KUKA KRL program: MyProgram_145().src

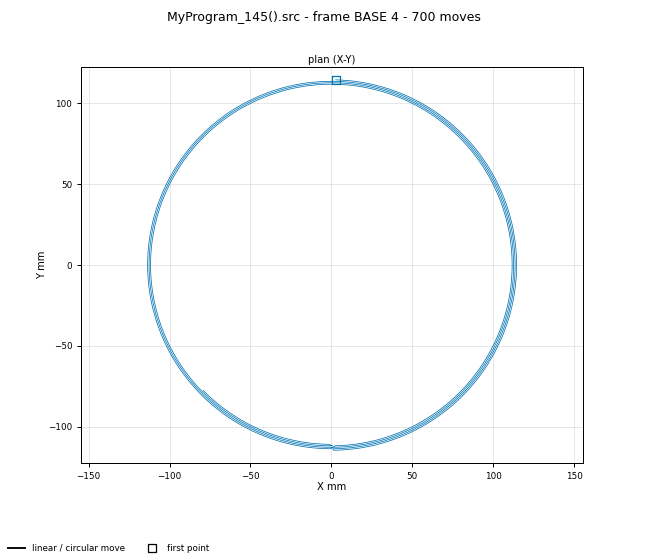
[picture p0: tool path of MyProgram_145().src in frame BASE 4, 700 of 700 moves have a stored position in this frame; points joined in program order, loops and branches not executed]
&ACCESS RVP
&REL 1
&PARAM TEMPLATE = C:\KRC\Roboter\Template\vorgabe
&PARAM EDITMASK = *
DEF MyProgram_145()
; ---- Setting reference (Base) ----
$BASE = BASE_DATA[4]

; --------------------------
; ---- Setting tool (TCP) ----
$TOOL = TOOL_DATA[3]
; --------------------------

$VEL.CP = VEL_APROX_PRINT
Startdeposition()
$VEL.CP = VEL_PRINT
LIN {X 2.5968,Y 114.457,Z 115,A 83.9175,B 24.9348,C -1.8654,E1 25.0049,E2 361.9885} C_DIS
LIN {X 5.4049,Y 114.3588,Z 115,A 82.5188,B 24.9348,C -1.8658,E1 25.0088,E2 363.3858} C_DIS
LIN {X 8.2098,Y 114.1917,Z 115,A 81.1109,B 24.9348,C -1.8657,E1 25.0127,E2 364.7933} C_DIS
LIN {X 10.8808,Y 113.9678,Z 115,A 79.7631,B 24.9348,C -1.8653,E1 25.0164,E2 366.1413} C_DIS
LIN {X 13.803,Y 113.6514,Z 115,A 78.3057,B 24.9348,C -1.8656,E1 25.0205,E2 367.5968} C_DIS
LIN {X 16.588,Y 113.2784,Z 115,A 76.9003,B 24.9348,C -1.8653,E1 25.0244,E2 369.0018} C_DIS
LIN {X 19.573,Y 112.8021,Z 115,A 75.3885,B 24.9348,C -1.8648,E1 25.0285,E2 370.5133} C_DIS
LIN {X 22.3354,Y 112.2877,Z 115,A 73.9836,B 24.9348,C -1.8643,E1 25.0324,E2 371.9177} C_DIS
LIN {X 25.0844,Y 111.7058,Z 115,A 72.5789,B 24.9348,C -1.8636,E1 25.0362,E2 373.3222} C_DIS
LIN {X 27.4876,Y 111.1372,Z 115,A 71.3329,B 24.935,C -1.8625,E1 25.0396,E2 374.569} C_DIS
LIN {X 30.3297,Y 110.3959,Z 115,A 69.8972,B 24.935,C -1.863,E1 25.0434,E2 376.0011} C_DIS
LIN {X 33.234,Y 109.5578,Z 115,A 68.3663,B 24.935,C -1.8611,E1 25.0476,E2 377.534} C_DIS
LIN {X 35.7101,Y 108.7747,Z 115,A 67.0558,B 24.9352,C -1.8596,E1 25.051,E2 378.8456} C_DIS
LIN {X 38.5697,Y 107.7951,Z 115,A 65.5589,B 24.9352,C -1.8589,E1 25.055,E2 380.3411} C_DIS
LIN {X 41.0044,Y 106.8915,Z 115,A 64.249,B 24.9353,C -1.8573,E1 25.0584,E2 381.6521} C_DIS
LIN {X 43.8125,Y 105.7727,Z 115,A 62.7522,B 24.9354,C -1.8564,E1 25.0623,E2 383.1476} C_DIS
LIN {X 46.3951,Y 104.6657,Z 115,A 61.3494,B 24.9355,C -1.855,E1 25.0659,E2 384.5503} C_DIS
LIN {X 48.9498,Y 103.4955,Z 115,A 59.9466,B 24.9356,C -1.8534,E1 25.0694,E2 385.9532} C_DIS
LIN {X 51.4749,Y 102.2631,Z 115,A 58.5442,B 24.9357,C -1.8518,E1 25.0729,E2 387.3557} C_DIS
LIN {X 53.9691,Y 100.969,Z 115,A 57.142,B 24.9358,C -1.8501,E1 25.0764,E2 388.7579} C_DIS
LIN {X 56.2448,Y 99.718,Z 115,A 55.8337,B 24.936,C -1.8479,E1 25.0796,E2 390.0676} C_DIS
LIN {X 58.8584,Y 98.1993,Z 115,A 54.3385,B 24.936,C -1.8464,E1 25.0832,E2 391.5617} C_DIS
LIN {X 60.7218,Y 97.0556,Z 115,A 53.1864,B 24.9364,C -1.8422,E1 25.0859,E2 392.7202} C_DIS
LIN {X 63.1456,Y 95.4964,Z 115,A 51.74,B 24.9366,C -1.8397,E1 25.0893,E2 394.1677} C_DIS
LIN {X 65.9229,Y 93.6033,Z 115,A 50.1344,B 24.9366,C -1.8403,E1 25.093,E2 395.7666} C_DIS
LIN {X 67.7672,Y 92.2743,Z 115,A 48.9337,B 24.9369,C -1.8355,E1 25.0957,E2 396.9743} C_DIS
LIN {X 70.2677,Y 90.3858,Z 115,A 47.4387,B 24.9369,C -1.8359,E1 25.099,E2 398.4629} C_DIS
LIN {X 72.3157,Y 88.7549,Z 115,A 46.1117,B 24.937,C -1.8327,E1 25.1019,E2 399.7924} C_DIS
LIN {X 74.3549,Y 87.0533,Z 115,A 44.7383,B 24.9374,C -1.8281,E1 25.1048,E2 401.1713} C_DIS
LIN {X 76.7265,Y 84.9717,Z 115,A 43.2249,B 24.9374,C -1.8279,E1 25.108,E2 402.6792} C_DIS
LIN {X 78.9438,Y 82.9173,Z 115,A 41.7315,B 24.9375,C -1.8256,E1 25.111,E2 404.1719} C_DIS
LIN {X 80.9549,Y 80.9549,Z 115,A 40.332,B 24.9377,C -1.8229,E1 25.1138,E2 405.5719} C_DIS
LIN {X 82.7695,Y 79.0971,Z 115,A 39.038,B 24.9379,C -1.8203,E1 25.1163,E2 406.8664} C_DIS
LIN {X 84.6857,Y 77.0421,Z 115,A 37.6386,B 24.9381,C -1.8174,E1 25.119,E2 408.2664} C_DIS
LIN {X 86.691,Y 74.7802,Z 115,A 36.1336,B 24.9383,C -1.8143,E1 25.1217,E2 409.7721} C_DIS
LIN {X 88.5001,Y 72.6301,Z 115,A 34.7343,B 24.9385,C -1.8113,E1 25.1242,E2 411.1721} C_DIS
LIN {X 90.1238,Y 70.6034,Z 115,A 33.4288,B 24.9387,C -1.8079,E1 25.1265,E2 412.4795} C_DIS
LIN {X 91.9573,Y 68.2002,Z 115,A 31.9366,B 24.9389,C -1.805,E1 25.129,E2 413.9712} C_DIS
LIN {X 93.6033,Y 65.9229,Z 115,A 30.5381,B 24.9391,C -1.8018,E1 25.1313,E2 415.3705} C_DIS
LIN {X 95.1929,Y 63.6059,Z 115,A 29.1395,B 24.9394,C -1.7986,E1 25.1335,E2 416.7699} C_DIS
LIN {X 96.3998,Y 61.7576,Z 115,A 27.9818,B 24.9397,C -1.7933,E1 25.1352,E2 417.9342} C_DIS
LIN {X 98.1993,Y 58.8584,Z 115,A 26.3429,B 24.9398,C -1.7918,E1 25.1376,E2 419.5682} C_DIS
LIN {X 99.5594,Y 56.5259,Z 115,A 24.9959,B 24.9401,C -1.7884,E1 25.1395,E2 420.9165} C_DIS
LIN {X 100.7076,Y 54.4511,Z 115,A 23.7501,B 24.9405,C -1.7824,E1 25.1412,E2 422.1698} C_DIS
LIN {X 102.1662,Y 51.6645,Z 115,A 22.2423,B 24.9405,C -1.7811,E1 25.1431,E2 423.6728} C_DIS
LIN {X 103.4955,Y 48.9497,Z 115,A 20.7513,B 24.9408,C -1.7777,E1 25.1449,E2 425.1636} C_DIS
LIN {X 104.5678,Y 46.6123,Z 115,A 19.4703,B 24.941,C -1.7743,E1 25.1464,E2 426.4457} C_DIS
LIN {X 105.7727,Y 43.8125,Z 115,A 17.9564,B 24.9413,C -1.7704,E1 25.148,E2 427.9606} C_DIS
LIN {X 106.8161,Y 41.2035,Z 115,A 16.5591,B 24.9415,C -1.7667,E1 25.1495,E2 429.3589} C_DIS
LIN {X 107.7951,Y 38.5697,Z 115,A 15.1617,B 24.9418,C -1.7629,E1 25.1508,E2 430.7574} C_DIS
LIN {X 108.5808,Y 36.2934,Z 115,A 13.9239,B 24.9421,C -1.7578,E1 25.1519,E2 432.0003} C_DIS
LIN {X 109.4947,Y 33.4374,Z 115,A 12.4606,B 24.9423,C -1.7549,E1 25.1531,E2 433.462} C_DIS
LIN {X 110.3313,Y 30.5674,Z 115,A 10.9865,B 24.9425,C -1.7513,E1 25.1543,E2 434.9361} C_DIS
LIN {X 111.0565,Y 27.8182,Z 115,A 9.5735,B 24.9428,C -1.7474,E1 25.1552,E2 436.3502} C_DIS
LIN {X 111.6579,Y 25.2918,Z 115,A 8.2822,B 24.943,C -1.7437,E1 25.1561,E2 437.6427} C_DIS
LIN {X 112.2877,Y 22.3354,Z 115,A 6.7797,B 24.9433,C -1.7394,E1 25.1569,E2 439.1466} C_DIS
LIN {X 112.8021,Y 19.573,Z 115,A 5.3829,B 24.9436,C -1.7354,E1 25.1576,E2 440.5446} C_DIS
LIN {X 113.2159,Y 17.0092,Z 115,A 4.0794,B 24.9438,C -1.7311,E1 25.1582,E2 441.8506} C_DIS
LIN {X 113.6266,Y 14.0145,Z 115,A 2.5896,B 24.9441,C -1.7273,E1 25.1587,E2 443.3406} C_DIS
LIN {X 113.9363,Y 11.2217,Z 115,A 1.193,B 24.9443,C -1.7233,E1 25.1591,E2 444.7385} C_DIS
LIN {X 114.1348,Y 8.9554,Z 115,A 0.0174,B 24.9447,C -1.7179,E1 25.1594,E2 445.9198} C_DIS
LIN {X 114.3379,Y 5.8302,Z 115,A -1.5068,B 24.9449,C -1.7148,E1 25.1596,E2 447.4422} C_DIS
LIN {X 114.4466,Y 3.0225,Z 115,A -2.9032,B 24.9452,C -1.7107,E1 25.1598,E2 448.8399} C_DIS
LIN {X 114.4869,Y 0,Z 115,A -4.3693,B 24.9453,C -1.708,E1 25.1598,E2 450.3038} C_DIS
LIN {X 114.4625,Y -2.2993,Z 115,A -5.5879,B 24.9458,C -1.7011,E1 25.1598,E2 451.5314} C_DIS
LIN {X 114.3588,Y -5.4049,Z 115,A -7.0927,B 24.9459,C -1.6983,E1 25.1596,E2 453.0337} C_DIS
LIN {X 114.1917,Y -8.2098,Z 115,A -8.4892,B 24.9462,C -1.6942,E1 25.1593,E2 454.4317} C_DIS
LIN {X 113.9363,Y -11.2217,Z 115,A -9.9788,B 24.9465,C -1.6903,E1 25.1589,E2 455.9216} C_DIS
LIN {X 113.6693,Y -13.6499,Z 115,A -11.1698,B 24.9466,C -1.6878,E1 25.1585,E2 457.1114} C_DIS
LIN {X 113.2484,Y -16.7988,Z 115,A -12.772,B 24.947,C -1.6821,E1 25.1579,E2 458.7177} C_DIS
LIN {X 112.8021,Y -19.573,Z 115,A -14.1682,B 24.9472,C -1.678,E1 25.1573,E2 460.1154} C_DIS
LIN {X 112.328,Y -22.1263,Z 115,A -15.4716,B 24.9475,C -1.6736,E1 25.1566,E2 461.4214} C_DIS
LIN {X 111.7058,Y -25.0844,Z 115,A -16.9615,B 24.9478,C -1.6698,E1 25.1557,E2 462.9117} C_DIS
LIN {X 111.0565,Y -27.8182,Z 115,A -18.358,B 24.948,C -1.6657,E1 25.1548,E2 464.3097} C_DIS
LIN {X 110.3959,Y -30.3297,Z 115,A -19.6489,B 24.9482,C -1.662,E1 25.1539,E2 465.6021} C_DIS
LIN {X 109.6183,Y -33.0299,Z 115,A -21.058,B 24.9485,C -1.6574,E1 25.1527,E2 467.014} C_DIS
LIN {X 108.7092,Y -35.9127,Z 115,A -22.5483,B 24.9488,C -1.6536,E1 25.1515,E2 468.5046} C_DIS
LIN {X 107.7951,Y -38.5697,Z 115,A -23.9448,B 24.949,C -1.6496,E1 25.1502,E2 469.9027} C_DIS
LIN {X 106.8915,Y -41.0044,Z 115,A -25.236,B 24.9492,C -1.646,E1 25.1489,E2 471.1953} C_DIS
LIN {X 105.7727,Y -43.8125,Z 115,A -26.7388,B 24.9495,C -1.6417,E1 25.1473,E2 472.6998} C_DIS
LIN {X 104.6657,Y -46.3951,Z 115,A -28.1358,B 24.9497,C -1.6379,E1 25.1458,E2 474.0983} C_DIS
LIN {X 103.4955,Y -48.9497,Z 115,A -29.5329,B 24.95,C -1.634,E1 25.1441,E2 475.497} C_DIS
LIN {X 102.3577,Y -51.2841,Z 115,A -30.8241,B 24.9502,C -1.6305,E1 25.1425,E2 476.7895} C_DIS
LIN {X 101.0683,Y -53.7807,Z 115,A -32.234,B 24.9505,C -1.6261,E1 25.1407,E2 478.2023} C_DIS
LIN {X 99.718,Y -56.2448,Z 115,A -33.6189,B 24.9506,C -1.623,E1 25.1388,E2 479.5875} C_DIS
LIN {X 98.1993,Y -58.8584,Z 115,A -35.1221,B 24.9509,C -1.619,E1 25.1367,E2 481.0923} C_DIS
LIN {X 96.8381,Y -61.07,Z 115,A -36.4264,B 24.9511,C -1.615,E1 25.1347,E2 482.3993} C_DIS
LIN {X 95.3102,Y -63.4281,Z 115,A -37.8117,B 24.9513,C -1.612,E1 25.1326,E2 483.7849} C_DIS
LIN {X 93.6033,Y -65.9229,Z 115,A -39.3154,B 24.9515,C -1.6081,E1 25.1302,E2 485.2903} C_DIS
LIN {X 92.0831,Y -68.0284,Z 115,A -40.6198,B 24.9518,C -1.6044,E1 25.1281,E2 486.5972} C_DIS
LIN {X 90.3858,Y -70.2677,Z 115,A -42.0057,B 24.9519,C -1.6015,E1 25.1257,E2 487.9834} C_DIS
LIN {X 88.6342,Y -72.4647,Z 115,A -43.4037,B 24.9521,C -1.5981,E1 25.1233,E2 489.3829} C_DIS
LIN {X 86.691,Y -74.7802,Z 115,A -44.9079,B 24.9524,C -1.5945,E1 25.1205,E2 490.8887} C_DIS
LIN {X 84.9717,Y -76.7265,Z 115,A -46.2006,B 24.9525,C -1.5915,E1 25.1181,E2 492.1827} C_DIS
LIN {X 82.9173,Y -78.9438,Z 115,A -47.7052,B 24.9527,C -1.588,E1 25.1153,E2 493.689} C_DIS
LIN {X 80.9549,Y -80.9549,Z 115,A -49.104,B 24.9529,C -1.5849,E1 25.1125,E2 495.0892} C_DIS
LIN {X 78.9438,Y -82.9173,Z 115,A -50.503,B 24.9531,C -1.5818,E1 25.1097,E2 496.4897} C_DIS
LIN {X 76.8852,Y -84.8297,Z 115,A -51.9019,B 24.9533,C -1.5788,E1 25.1068,E2 497.8901} C_DIS
LIN {X 74.9406,Y -86.5509,Z 115,A -53.1952,B 24.9535,C -1.5761,E1 25.1041,E2 499.1846} C_DIS
LIN {X 72.6302,Y -88.5001,Z 115,A -54.701,B 24.9536,C -1.573,E1 25.1009,E2 500.6919} C_DIS
LIN {X 70.4364,Y -90.2559,Z 115,A -56.1002,B 24.9538,C -1.5702,E1 25.0978,E2 502.0925} C_DIS
LIN {X 68.3704,Y -91.8294,Z 115,A -57.4068,B 24.954,C -1.5671,E1 25.0949,E2 503.4016} C_DIS
LIN {X 66.0962,Y -93.4796,Z 115,A -58.7941,B 24.9541,C -1.5651,E1 25.0917,E2 504.7889} C_DIS
LIN {X 63.6059,Y -95.1929,Z 115,A -60.3003,B 24.9543,C -1.5623,E1 25.0882,E2 506.2966} C_DIS
LIN {X 61.4298,Y -96.6102,Z 115,A -61.6073,B 24.9544,C -1.5594,E1 25.0852,E2 507.6061} C_DIS
LIN {X 58.8584,Y -98.1993,Z 115,A -63.1013,B 24.9546,C -1.5574,E1 25.0816,E2 509.1002} C_DIS
LIN {X 56.4307,Y -99.6142,Z 115,A -64.5018,B 24.9546,C -1.5551,E1 25.0782,E2 510.5019} C_DIS
LIN {X 52.726,Y -101.6237,Z 115,A -66.6037,B 24.9549,C -1.5518,E1 25.073,E2 512.6057} C_DIS
LIN {X 50.2161,Y -102.8871,Z 115,A -68.0047,B 24.955,C -1.5497,E1 25.0695,E2 514.0079} C_DIS
LIN {X 47.8691,Y -103.9986,Z 115,A -69.3001,B 24.9551,C -1.5478,E1 25.0662,E2 515.3044} C_DIS
LIN {X 45.3024,Y -105.142,Z 115,A -70.7144,B 24.9553,C -1.5453,E1 25.0626,E2 516.7212} C_DIS
LIN {X 42.7084,Y -106.2221,Z 115,A -72.1165,B 24.9553,C -1.5435,E1 25.059,E2 518.1244} C_DIS
LIN {X 39.8896,Y -107.3137,Z 115,A -73.6122,B 24.9554,C -1.5421,E1 25.0551,E2 519.62} C_DIS
LIN {X 37.4449,Y -108.1898,Z 115,A -74.9078,B 24.9555,C -1.5407,E1 25.0517,E2 520.9166} C_DIS
LIN {X 34.7785,Y -109.0762,Z 115,A -76.3108,B 24.9556,C -1.5391,E1 25.0479,E2 522.3206} C_DIS
LIN {X 31.887,Y -109.9574,Z 115,A -77.8197,B 24.9557,C -1.5375,E1 25.0439,E2 523.8307} C_DIS
LIN {X 29.179,Y -110.7068,Z 115,A -79.2228,B 24.9557,C -1.5361,E1 25.0401,E2 525.2348} C_DIS
LIN {X 26.6601,Y -111.3391,Z 115,A -80.5196,B 24.9559,C -1.535,E1 25.0366,E2 526.5324} C_DIS
LIN {X 23.9197,Y -111.9598,Z 115,A -81.923,B 24.9559,C -1.5338,E1 25.0328,E2 527.9368} C_DIS
LIN {X 20.9558,Y -112.5534,Z 115,A -83.4333,B 24.9559,C -1.5326,E1 25.0286,E2 529.4481} C_DIS
LIN {X 18.3973,Y -112.9986,Z 115,A -84.7433,B 24.9561,C -1.5311,E1 25.025,E2 530.7601} C_DIS
LIN {X 15.6186,Y -113.4161,Z 115,A -86.1372,B 24.9561,C -1.5307,E1 25.0212,E2 532.1538} C_DIS
LIN {X 12.6191,Y -113.79,Z 115,A -87.6457,B 24.9561,C -1.53,E1 25.017,E2 533.663} C_DIS
LIN {X 10.0348,Y -114.0459,Z 115,A -88.9441,B 24.9561,C -1.5293,E1 25.0134,E2 534.9621} C_DIS
LIN {X 7.0205,Y -114.2721,Z 115,A -90.4554,B 24.9562,C -1.5287,E1 25.0091,E2 536.4742} C_DIS
LIN {X 4.214,Y -114.41,Z 115,A -91.8604,B 24.9562,C -1.5282,E1 25.0052,E2 537.8799} C_DIS
LIN {X 1.4049,Y -114.479,Z 115,A -93.2656,B 24.9562,C -1.5279,E1 25.0013,E2 539.2858} C_DIS
LIN {X 1.4049,Y -114.479,Z 115,A -93.2656,B 24.9562,C -1.5279,E1 25.0013,E2 539.2858} C_DIS
Enddeposition()
LIN {X 0.793,Y -113.5682,Z 115,A -93.0605,B 24.954,C -1.5662,E1 25.0021,E2 538.9899} C_DIS
Startdeposition()
$VEL.CP = VEL_PRINT
LIN {X 3.5216,Y -113.5178,Z 115,A -91.1293,B 24.9526,C -1.591,E1 25.0077,E2 537.0003} C_DIS
LIN {X 6.9982,Y -113.3576,Z 115,A -89.1991,B 24.9521,C -1.5995,E1 25.0131,E2 535.0508} C_DIS
LIN {X 11.2037,Y -113.0202,Z 115,A -87.4324,B 24.953,C -1.5845,E1 25.0179,E2 533.3206} C_DIS
LIN {X 15.2462,Y -112.546,Z 115,A -84.7536,B 24.9512,C -1.6138,E1 25.0255,E2 530.5747} C_DIS
LIN {X 20.5071,Y -111.7064,Z 115,A -82.954,B 24.9535,C -1.5762,E1 25.0302,E2 528.866} C_DIS
LIN {X 23.3283,Y -111.1518,Z 115,A -81.5254,B 24.9535,C -1.5765,E1 25.0341,E2 527.4385} C_DIS
LIN {X 26.2423,Y -110.5012,Z 115,A -79.8314,B 24.9529,C -1.5863,E1 25.0388,E2 525.7237} C_DIS
LIN {X 30.1207,Y -109.5066,Z 115,A -78.0115,B 24.9533,C -1.5795,E1 25.0437,E2 523.9227} C_DIS
LIN {X 33.4764,Y -108.5267,Z 115,A -76.2704,B 24.9532,C -1.5806,E1 25.0483,E2 522.1821} C_DIS
LIN {X 36.5165,Y -107.5421,Z 115,A -74.492,B 24.9526,C -1.59,E1 25.0531,E2 520.3848} C_DIS
LIN {X 41.5359,Y -105.7046,Z 115,A -71.5463,B 24.9517,C -1.605,E1 25.0608,E2 517.41} C_DIS
LIN {X 44.5412,Y -104.4748,Z 115,A -70.157,B 24.9523,C -1.5961,E1 25.0644,E2 516.045} C_DIS
LIN {X 48.1845,Y -102.8446,Z 115,A -68.3364,B 24.9526,C -1.5905,E1 25.0689,E2 514.2422} C_DIS
LIN {X 51.1511,Y -101.4032,Z 115,A -66.6992,B 24.9526,C -1.592,E1 25.073,E2 512.6057} C_DIS
LIN {X 54.0223,Y -99.9014,Z 115,A -64.9679,B 24.9521,C -1.5993,E1 25.0773,E2 510.8623} C_DIS
LIN {X 56.7874,Y -98.3561,Z 115,A -63.465,B 24.9521,C -1.5978,E1 25.081,E2 509.3673} C_DIS
LIN {X 59.5307,Y -96.7221,Z 115,A -61.5707,B 24.9512,C -1.6138,E1 25.0856,E2 507.4412} C_DIS
LIN {X 63.3856,Y -94.2395,Z 115,A -59.4229,B 24.9514,C -1.6108,E1 25.0905,E2 505.3076} C_DIS
LIN {X 66.4794,Y -92.0846,Z 115,A -57.6419,B 24.9514,C -1.6092,E1 25.0946,E2 503.5366} C_DIS
LIN {X 69.0541,Y -90.1684,Z 115,A -56.0169,B 24.9513,C -1.6129,E1 25.0982,E2 501.9086} C_DIS
LIN {X 71.7186,Y -88.0636,Z 115,A -54.1829,B 24.9507,C -1.6223,E1 25.1022,E2 500.0594} C_DIS
LIN {X 74.7011,Y -85.5478,Z 115,A -52.3131,B 24.9507,C -1.6223,E1 25.1062,E2 498.1969} C_DIS
LIN {X 77.2866,Y -83.2222,Z 115,A -50.4101,B 24.95,C -1.6332,E1 25.1101,E2 496.2757} C_DIS
LIN {X 79.9158,Y -80.698,Z 115,A -48.7126,B 24.9501,C -1.6312,E1 25.1135,E2 494.5901} C_DIS
LIN {X 82.5394,Y -78.0129,Z 115,A -46.8265,B 24.9499,C -1.6356,E1 25.1171,E2 492.7018} C_DIS
LIN {X 84.8762,Y -75.4643,Z 115,A -45.1773,B 24.9499,C -1.6356,E1 25.1202,E2 491.0597} C_DIS
LIN {X 87.1423,Y -72.8355,Z 115,A -43.3428,B 24.9493,C -1.6441,E1 25.1236,E2 489.2136} C_DIS
LIN {X 89.4592,Y -69.972,Z 115,A -41.4045,B 24.9488,C -1.6528,E1 25.1269,E2 487.2639} C_DIS
LIN {X 91.6183,Y -67.1176,Z 115,A -39.7048,B 24.9488,C -1.6529,E1 25.1298,E2 485.5722} C_DIS
LIN {X 93.3527,Y -64.6838,Z 115,A -38.187,B 24.9485,C -1.6576,E1 25.1322,E2 484.0508} C_DIS
LIN {X 95.0825,Y -62.1147,Z 115,A -36.7548,B 24.9486,C -1.6559,E1 25.1344,E2 482.6296} C_DIS
LIN {X 96.7961,Y -59.4091,Z 115,A -34.9771,B 24.9479,C -1.6681,E1 25.137,E2 480.8321} C_DIS
LIN {X 98.7922,Y -56.0286,Z 115,A -32.9319,B 24.9473,C -1.677,E1 25.1399,E2 478.7767} C_DIS
LIN {X 100.7462,Y -52.4329,Z 115,A -31.1232,B 24.9477,C -1.6712,E1 25.1423,E2 476.9912} C_DIS
LIN {X 102.1239,Y -49.6963,Z 115,A -29.3014,B 24.9466,C -1.6887,E1 25.1445,E2 475.1377} C_DIS
LIN {X 104.0236,Y -45.5832,Z 115,A -27.1729,B 24.9466,C -1.6884,E1 25.147,E2 473.0215} C_DIS
LIN {X 105.434,Y -42.2225,Z 115,A -25.4888,B 24.9466,C -1.6868,E1 25.1487,E2 471.3503} C_DIS
LIN {X 106.9636,Y -38.1818,Z 115,A -23.3424,B 24.9463,C -1.6921,E1 25.1508,E2 469.2036} C_DIS
LIN {X 108.0365,Y -35.0258,Z 115,A -21.6182,B 24.9459,C -1.6994,E1 25.1524,E2 467.4719} C_DIS
LIN {X 109.0809,Y -31.6306,Z 115,A -19.8607,B 24.9456,C -1.7035,E1 25.1538,E2 465.7149} C_DIS
LIN {X 110.0465,Y -28.0802,Z 115,A -17.9109,B 24.945,C -1.7138,E1 25.1552,E2 463.7518} C_DIS
LIN {X 110.7958,Y -24.9668,Z 115,A -16.4113,B 24.945,C -1.7136,E1 25.1561,E2 462.2615} C_DIS
LIN {X 111.3099,Y -22.5582,Z 115,A -15.0009,B 24.9442,C -1.7255,E1 25.1569,E2 460.8313} C_DIS
LIN {X 112.007,Y -18.7917,Z 115,A -13.1014,B 24.9439,C -1.7302,E1 25.1578,E2 458.9318} C_DIS
LIN {X 112.5769,Y -15.0105,Z 115,A -11.227,B 24.9437,C -1.7339,E1 25.1586,E2 457.0597} C_DIS
LIN {X 113.2173,Y -8.9741,Z 115,A -8.4018,B 24.9437,C -1.7327,E1 25.1594,E2 454.2539} C_DIS
LIN {X 113.3861,Y -6.5058,Z 115,A -6.9816,B 24.9429,C -1.7448,E1 25.1596,E2 452.8136} C_DIS
LIN {X 113.5363,Y -2.917,Z 115,A -4.3528,B 24.94,C -1.7892,E1 25.1598,E2 450.0958} C_DIS
LIN {X 113.5471,Y 2.4173,Z 115,A -2.7769,B 24.9429,C -1.7455,E1 25.1598,E2 448.6324} C_DIS
LIN {X 113.2765,Y 8.2121,Z 115,A 0.436,B 24.9414,C -1.7683,E1 25.1593,E2 445.3849} C_DIS
LIN {X 112.7669,Y 13.5054,Z 115,A 2.9476,B 24.9414,C -1.7689,E1 25.1586,E2 442.8867} C_DIS
LIN {X 112.3726,Y 16.4724,Z 115,A 4.6823,B 24.9403,C -1.7842,E1 25.1579,E2 441.1262} C_DIS
LIN {X 111.7823,Y 20.0848,Z 115,A 6.415,B 24.9403,C -1.7847,E1 25.157,E2 439.4023} C_DIS
LIN {X 111.1336,Y 23.4171,Z 115,A 8.0257,B 24.9403,C -1.7853,E1 25.1561,E2 437.7996} C_DIS
LIN {X 110.3519,Y 26.8541,Z 115,A 9.8366,B 24.9398,C -1.7924,E1 25.155,E2 435.9825} C_DIS
LIN {X 109.5022,Y 30.1371,Z 115,A 11.4761,B 24.9397,C -1.7944,E1 25.1538,E2 434.3479} C_DIS
LIN {X 108.7794,Y 32.6475,Z 115,A 12.7391,B 24.9396,C -1.7959,E1 25.1528,E2 433.0885} C_DIS
LIN {X 107.8376,Y 35.64,Z 115,A 14.5381,B 24.9385,C -1.8107,E1 25.1513,E2 431.2648} C_DIS
LIN {X 106.4359,Y 39.6278,Z 115,A 17.2456,B 24.9363,C -1.8439,E1 25.1486,E2 428.4941} C_DIS
LIN {X 104.7174,Y 43.9657,Z 115,A 19.028,B 24.9376,C -1.8241,E1 25.1467,E2 426.7682} C_DIS
LIN {X 102.9135,Y 48.0365,Z 115,A 21.1776,B 24.9375,C -1.8261,E1 25.1443,E2 424.6255} C_DIS
LIN {X 101.1901,Y 51.568,Z 115,A 23.0853,B 24.9373,C -1.8282,E1 25.1419,E2 422.7229} C_DIS
LIN {X 99.69,Y 54.4122,Z 115,A 24.8126,B 24.9367,C -1.8376,E1 25.1396,E2 420.9827} C_DIS
LIN {X 97.6246,Y 58.0362,Z 115,A 26.897,B 24.9364,C -1.8423,E1 25.1367,E2 418.8978} C_DIS
LIN {X 95.8022,Y 60.9983,Z 115,A 28.5559,B 24.9364,C -1.8426,E1 25.1342,E2 417.2468} C_DIS
LIN {X 93.9892,Y 63.7552,Z 115,A 30.2244,B 24.936,C -1.8471,E1 25.1316,E2 415.5759} C_DIS
LIN {X 91.8075,Y 66.8592,Z 115,A 32.1034,B 24.9358,C -1.8503,E1 25.1286,E2 413.6984} C_DIS
LIN {X 89.2992,Y 70.1743,Z 115,A 34.2418,B 24.9353,C -1.8573,E1 25.1249,E2 411.5536} C_DIS
LIN {X 86.9459,Y 73.0718,Z 115,A 35.9983,B 24.9354,C -1.856,E1 25.1218,E2 409.8084} C_DIS
LIN {X 85.1265,Y 75.1835,Z 115,A 37.8359,B 24.9338,C -1.8789,E1 25.1183,E2 407.9248} C_DIS
LIN {X 82.9605,Y 77.5651,Z 115,A 38.8497,B 24.9355,C -1.8548,E1 25.1165,E2 406.9725} C_DIS
LIN {X 81.1764,Y 79.4315,Z 115,A 40.4567,B 24.9343,C -1.8714,E1 25.1133,E2 405.333} C_DIS
LIN {X 78.5548,Y 82.0241,Z 115,A 42.3562,B 24.9339,C -1.8772,E1 25.1095,E2 403.4279} C_DIS
LIN {X 76.3037,Y 84.1241,Z 115,A 43.7221,B 24.9343,C -1.8719,E1 25.1068,E2 402.0801} C_DIS
LIN {X 74.383,Y 85.8256,Z 115,A 44.9967,B 24.9342,C -1.8735,E1 25.1041,E2 400.8066} C_DIS
LIN {X 71.7145,Y 88.067,Z 115,A 46.7426,B 24.934,C -1.8764,E1 25.1003,E2 399.0607} C_DIS
LIN {X 69.2353,Y 90.0287,Z 115,A 48.4361,B 24.9335,C -1.8838,E1 25.0966,E2 397.3559} C_DIS
LIN {X 66.661,Y 91.9526,Z 115,A 50.3108,B 24.9325,C -1.898,E1 25.0923,E2 395.4542} C_DIS
LIN {X 61.7781,Y 95.3017,Z 115,A 52.8464,B 24.9336,C -1.8826,E1 25.0865,E2 392.9634} C_DIS
LIN {X 59.1525,Y 96.9521,Z 115,A 54.5541,B 24.9329,C -1.8915,E1 25.0824,E2 391.2403} C_DIS
LIN {X 55.9057,Y 98.8616,Z 115,A 56.5872,B 24.9323,C -1.9001,E1 25.0775,E2 389.1929} C_DIS
LIN {X 52.271,Y 100.8308,Z 115,A 59.5639,B 24.9292,C -1.9428,E1 25.0699,E2 386.1234} C_DIS
LIN {X 46.742,Y 103.5079,Z 115,A 61.52,B 24.9326,C -1.8955,E1 25.0652,E2 384.2843} C_DIS
LIN {X 44.5083,Y 104.4887,Z 115,A 62.9545,B 24.9319,C -1.9058,E1 25.0615,E2 382.8287} C_DIS
LIN {X 41.3685,Y 105.7703,Z 115,A 64.594,B 24.932,C -1.9044,E1 25.0572,E2 381.1963} C_DIS
LIN {X 38.3334,Y 106.9094,Z 115,A 66.2855,B 24.9317,C -1.9084,E1 25.0528,E2 379.4989} C_DIS
LIN {X 35.2317,Y 107.9699,Z 115,A 67.8646,B 24.9319,C -1.9065,E1 25.0486,E2 377.9273} C_DIS
LIN {X 32.0949,Y 108.9433,Z 115,A 69.5697,B 24.9316,C -1.9098,E1 25.044,E2 376.2173} C_DIS
LIN {X 28.9079,Y 109.8337,Z 115,A 71.0773,B 24.932,C -1.9038,E1 25.04,E2 374.7263} C_DIS
LIN {X 26.7238,Y 110.3837,Z 115,A 72.3303,B 24.9316,C -1.9096,E1 25.0366,E2 373.4614} C_DIS
LIN {X 23.5774,Y 111.1,Z 115,A 73.847,B 24.9319,C -1.9056,E1 25.0325,E2 371.9563} C_DIS
LIN {X 19.753,Y 111.842,Z 115,A 75.8698,B 24.9317,C -1.9089,E1 25.0269,E2 369.928} C_DIS
LIN {X 16.0692,Y 112.4299,Z 115,A 78.0906,B 24.9306,C -1.9241,E1 25.0207,E2 367.6731} C_DIS
LIN {X 11.714,Y 112.9667,Z 115,A 80.2368,B 24.9308,C -1.9215,E1 25.0147,E2 365.5345} C_DIS
LIN {X 7.3617,Y 113.3339,Z 115,A 82.1205,B 24.9318,C -1.9079,E1 25.0096,E2 363.6841} C_DIS
LIN {X 1.1044,Y 113.5677,Z 115,A 85.1447,B 24.9322,C -1.9018,E1 25.0012,E2 360.6751} C_DIS
LIN {X -5.6869,Y 113.4314,Z 115,A 88.6544,B 24.932,C -1.9042,E1 24.9914,E2 357.1591} C_DIS
LIN {X -12.5625,Y 112.8773,Z 115,A 92.1705,B 24.932,C -1.9041,E1 24.9816,E2 353.6418} C_DIS
LIN {X -15.4607,Y 112.5163,Z 115,A 93.7976,B 24.9316,C -1.9097,E1 24.977,E2 352.0001} C_DIS
LIN {X -18.9323,Y 111.9835,Z 115,A 95.4868,B 24.932,C -1.9049,E1 24.9724,E2 350.3206} C_DIS
LIN {X -22.6369,Y 111.2938,Z 115,A 97.4268,B 24.932,C -1.905,E1 24.9671,E2 348.3783} C_DIS
LIN {X -26.2566,Y 110.4977,Z 115,A 99.2119,B 24.9323,C -1.8998,E1 24.9623,E2 346.6034} C_DIS
LIN {X -29.7238,Y 109.6138,Z 115,A 101.1437,B 24.9321,C -1.9033,E1 24.957,E2 344.6604} C_DIS
LIN {X -33.7888,Y 108.4298,Z 115,A 103.2853,B 24.9322,C -1.9011,E1 24.9513,E2 342.5204} C_DIS
LIN {X -37.4761,Y 107.2112,Z 115,A 105.2615,B 24.9324,C -1.8994,E1 24.9461,E2 340.5444} C_DIS
LIN {X -41.4151,Y 105.752,Z 115,A 107.3253,B 24.9327,C -1.8943,E1 24.9407,E2 338.4885} C_DIS
LIN {X -45.2042,Y 104.1888,Z 115,A 109.2418,B 24.9334,C -1.885,E1 24.9358,E2 336.5895} C_DIS
LIN {X -47.5976,Y 103.1178,Z 115,A 110.6962,B 24.9331,C -1.8884,E1 24.9321,E2 335.1235} C_DIS
LIN {X -53.0774,Y 100.4067,Z 115,A 113.9148,B 24.9331,C -1.8889,E1 24.9241,E2 331.8953} C_DIS
LIN {X -56.5974,Y 98.4653,Z 115,A 115.8907,B 24.9335,C -1.8832,E1 24.9192,E2 329.9271} C_DIS
LIN {X -60.6035,Y 96.0529,Z 115,A 118.1284,B 24.9342,C -1.8738,E1 24.914,E2 327.7049} C_DIS
LIN {X -63.2127,Y 94.3565,Z 115,A 119.7424,B 24.9342,C -1.8725,E1 24.9102,E2 326.0885} C_DIS
LIN {X -65.9791,Y 92.4416,Z 115,A 121.5286,B 24.9342,C -1.8727,E1 24.9061,E2 324.2957} C_DIS
LIN {X -68.5003,Y 90.5899,Z 115,A 123.0471,B 24.9347,C -1.867,E1 24.9027,E2 322.7855} C_DIS
LIN {X -71.1466,Y 88.5272,Z 115,A 124.6224,B 24.9353,C -1.8585,E1 24.8993,E2 321.2245} C_DIS
LIN {X -72.8647,Y 87.118,Z 115,A 125.8209,B 24.9353,C -1.8592,E1 24.8967,E2 320.0198} C_DIS
LIN {X -74.7298,Y 85.5227,Z 115,A 127.2065,B 24.935,C -1.8623,E1 24.8937,E2 318.6213} C_DIS
LIN {X -77.3644,Y 83.1493,Z 115,A 129.0946,B 24.935,C -1.8621,E1 24.8899,E2 316.726} C_DIS
LIN {X -80.3903,Y 80.2273,Z 115,A 130.9762,B 24.936,C -1.8473,E1 24.8862,E2 314.8718} C_DIS
LIN {X -82.0223,Y 78.5568,Z 115,A 132.1783,B 24.9362,C -1.8454,E1 24.8838,E2 313.6692} C_DIS
LIN {X -83.6587,Y 76.8108,Z 115,A 133.5393,B 24.9359,C -1.8485,E1 24.8812,E2 312.2947} C_DIS
LIN {X -85.8919,Y 74.3071,Z 115,A 135.1233,B 24.9366,C -1.8398,E1 24.8783,E2 310.7243} C_DIS
LIN {X -88.1599,Y 71.5998,Z 115,A 137.0204,B 24.9366,C -1.8398,E1 24.8749,E2 308.8185} C_DIS
LIN {X -89.8764,Y 69.433,Z 115,A 138.4651,B 24.9366,C -1.838,E1 24.8725,E2 307.3712} C_DIS
LIN {X -92.3919,Y 66.0488,Z 115,A 140.5171,B 24.9373,C -1.8292,E1 24.8691,E2 305.3303} C_DIS
LIN {X -94.9972,Y 62.2441,Z 115,A 143.0368,B 24.9373,C -1.8304,E1 24.8651,E2 302.7951} C_DIS
LIN {X -97.6334,Y 58.0213,Z 115,A 145.5732,B 24.9376,C -1.8242,E1 24.8615,E2 300.2606} C_DIS
LIN {X -100.0382,Y 53.7701,Z 115,A 147.7983,B 24.9388,C -1.8074,E1 24.8585,E2 298.0637} C_DIS
LIN {X -101.6163,Y 50.7238,Z 115,A 149.5615,B 24.939,C -1.8035,E1 24.8563,E2 296.3004} C_DIS
LIN {X -103.0763,Y 47.6869,Z 115,A 151.224,B 24.9395,C -1.7969,E1 24.8543,E2 294.6446} C_DIS
LIN {X -104.5463,Y 44.3717,Z 115,A 153.4502,B 24.9388,C -1.8071,E1 24.8518,E2 292.3817} C_DIS
LIN {X -106.3238,Y 39.9255,Z 115,A 155.5265,B 24.9402,C -1.7861,E1 24.8497,E2 290.3439} C_DIS
LIN {X -107.4582,Y 36.7652,Z 115,A 157.8104,B 24.939,C -1.8043,E1 24.8476,E2 288.0036} C_DIS
LIN {X -108.6452,Y 33.0938,Z 115,A 159.1494,B 24.941,C -1.7739,E1 24.8465,E2 286.7293} C_DIS
LIN {X -109.4371,Y 30.3739,Z 115,A 160.9454,B 24.9404,C -1.7839,E1 24.8451,E2 284.899} C_DIS
LIN {X -110.3649,Y 26.8009,Z 115,A 162.5325,B 24.9415,C -1.7671,E1 24.8441,E2 283.3429} C_DIS
LIN {X -111.0575,Y 23.772,Z 115,A 164.0567,B 24.9419,C -1.7603,E1 24.8432,E2 281.8259} C_DIS
LIN {X -111.6428,Y 20.8559,Z 115,A 165.8197,B 24.9416,C -1.7659,E1 24.8422,E2 280.0392} C_DIS
LIN {X -112.1949,Y 17.6376,Z 115,A 167.2848,B 24.9424,C -1.7533,E1 24.8416,E2 278.5952} C_DIS
LIN {X -112.6393,Y 14.5283,Z 115,A 168.9357,B 24.9425,C -1.7508,E1 24.841,E2 276.9404} C_DIS
LIN {X -113.0125,Y 11.2767,Z 115,A 170.6947,B 24.9426,C -1.7497,E1 24.8404,E2 275.1735} C_DIS
LIN {X -113.2977,Y 7.8984,Z 115,A 172.3163,B 24.9432,C -1.7407,E1 24.8401,E2 273.5639} C_DIS
LIN {X -113.4806,Y 4.5744,Z 115,A 174.0587,B 24.9434,C -1.7377,E1 24.8399,E2 271.8181} C_DIS
LIN {X -113.5702,Y 0.7165,Z 115,A 176.0092,B 24.9438,C -1.7315,E1 24.8398,E2 269.8705} C_DIS
LIN {X -113.5239,Y -3.3225,Z 115,A 178.0504,B 24.9442,C -1.725,E1 24.8398,E2 267.8324} C_DIS
LIN {X -113.3332,Y -7.373,Z 115,A -179.933,B 24.9447,C -1.7173,E1 24.8402,E2 265.8222} C_DIS
LIN {X -113.0459,Y -10.9348,Z 115,A -178.1846,B 24.9452,C -1.7093,E1 24.8406,E2 264.0823} C_DIS
LIN {X -112.7864,Y -13.3391,Z 115,A -176.9395,B 24.9454,C -1.7064,E1 24.841,E2 262.8367} C_DIS
LIN {X -112.3452,Y -16.6648,Z 115,A -175.0424,B 24.9453,C -1.7092,E1 24.8418,E2 260.9217} C_DIS
LIN {X -111.8036,Y -19.9665,Z 115,A -173.4065,B 24.9457,C -1.7018,E1 24.8426,E2 259.2937} C_DIS
LIN {X -111.145,Y -23.3614,Z 115,A -171.6451,B 24.946,C -1.6969,E1 24.8435,E2 257.5334} C_DIS
LIN {X -110.3339,Y -26.9281,Z 115,A -169.8542,B 24.9465,C -1.6891,E1 24.8447,E2 255.7508} C_DIS
LIN {X -108.2801,Y -34.2719,Z 115,A -165.3888,B 24.9457,C -1.7021,E1 24.8483,E2 251.2286} C_DIS
LIN {X -106.9164,Y -38.3143,Z 115,A -163.9116,B 24.9478,C -1.6685,E1 24.8496,E2 249.8231} C_DIS
LIN {X -106.0683,Y -40.6001,Z 115,A -162.6951,B 24.9481,C -1.6643,E1 24.8507,E2 248.6097} C_DIS
LIN {X -105.2093,Y -42.7748,Z 115,A -161.472,B 24.9481,C -1.6626,E1 24.852,E2 247.3838} C_DIS
LIN {X -103.9172,Y -45.8273,Z 115,A -159.5857,B 24.948,C -1.6664,E1 24.8541,E2 245.4781} C_DIS
LIN {X -102.1287,Y -49.6863,Z 115,A -157.5633,B 24.9487,C -1.6553,E1 24.8565,E2 243.4711} C_DIS
LIN {X -100.0587,Y -53.7323,Z 115,A -155.2087,B 24.9489,C -1.6514,E1 24.8596,E2 241.1132} C_DIS
LIN {X -98.2969,Y -56.8904,Z 115,A -153.4798,B 24.9494,C -1.6426,E1 24.8619,E2 239.3962} C_DIS
LIN {X -96.9399,Y -59.1725,Z 115,A -152.0842,B 24.9495,C -1.6413,E1 24.864,E2 237.9965} C_DIS
LIN {X -95.405,Y -61.6172,Z 115,A -150.681,B 24.9499,C -1.6354,E1 24.8661,E2 236.6005} C_DIS
LIN {X -93.5701,Y -64.3709,Z 115,A -149.0489,B 24.9502,C -1.6296,E1 24.8686,E2 234.974} C_DIS
LIN {X -91.6717,Y -67.0446,Z 115,A -147.3589,B 24.9504,C -1.6269,E1 24.8714,E2 233.2822} C_DIS
LIN {X -89.4421,Y -69.9935,Z 115,A -145.5182,B 24.9507,C -1.6213,E1 24.8745,E2 231.446} C_DIS
LIN {X -87.9082,Y -71.9104,Z 115,A -144.2034,B 24.9507,C -1.6215,E1 24.8768,E2 230.1247} C_DIS
LIN {X -82.6332,Y -77.9132,Z 115,A -140.0978,B 24.9511,C -1.6152,E1 24.8845,E2 226.0156} C_DIS
LIN {X -79.9602,Y -80.6541,Z 115,A -138.1746,B 24.9514,C -1.6107,E1 24.8882,E2 224.0949} C_DIS
LIN {X -77.3906,Y -83.1246,Z 115,A -136.4031,B 24.9517,C -1.6059,E1 24.8918,E2 222.3276} C_DIS
LIN {X -75.264,Y -85.0556,Z 115,A -134.6048,B 24.951,C -1.6174,E1 24.8956,E2 220.4947} C_DIS
LIN {X -71.3739,Y -88.343,Z 115,A -132.2231,B 24.9517,C -1.6048,E1 24.9007,E2 218.134} C_DIS
LIN {X -68.7995,Y -90.3646,Z 115,A -130.7145,B 24.9523,C -1.5959,E1 24.904,E2 216.6412} C_DIS
LIN {X -66.1638,Y -92.3098,Z 115,A -128.9283,B 24.9521,C -1.5986,E1 24.9081,E2 214.8422} C_DIS
LIN {X -62.9128,Y -94.5563,Z 115,A -127.0919,B 24.9527,C -1.5888,E1 24.9123,E2 213.023} C_DIS
LIN {X -60.2009,Y -96.3044,Z 115,A -125.3035,B 24.9525,C -1.593,E1 24.9165,E2 211.2189} C_DIS
LIN {X -56.9594,Y -98.2573,Z 115,A -123.3295,B 24.9525,C -1.5929,E1 24.9213,E2 209.2391} C_DIS
LIN {X -53.7047,Y -100.0737,Z 115,A -121.6173,B 24.953,C -1.5833,E1 24.9254,E2 207.5449} C_DIS
LIN {X -51.5866,Y -101.1806,Z 115,A -120.4005,B 24.953,C -1.5822,E1 24.9284,E2 206.3273} C_DIS
LIN {X -48.617,Y -102.6424,Z 115,A -118.6129,B 24.953,C -1.5851,E1 24.933,E2 204.5281} C_DIS
LIN {X -44.9477,Y -104.3006,Z 115,A -116.4782,B 24.9528,C -1.5873,E1 24.9384,E2 202.3833} C_DIS
LIN {X -41.1917,Y -105.8398,Z 115,A -114.6699,B 24.9535,C -1.5751,E1 24.9431,E2 200.5999} C_DIS
LIN {X -38.275,Y -106.9307,Z 115,A -112.8673,B 24.953,C -1.5835,E1 24.9479,E2 198.7737} C_DIS
LIN {X -34.3497,Y -108.2552,Z 115,A -110.9785,B 24.9536,C -1.5733,E1 24.9528,E2 196.9058} C_DIS
LIN {X -31.768,Y -109.0403,Z 115,A -109.4647,B 24.9533,C -1.5789,E1 24.9569,E2 195.3762} C_DIS
LIN {X -28.3478,Y -109.9777,Z 115,A -107.7436,B 24.9535,C -1.5749,E1 24.9615,E2 193.662} C_DIS
LIN {X -24.9677,Y -110.7956,Z 115,A -105.8753,B 24.9533,C -1.5788,E1 24.9667,E2 191.7817} C_DIS
LIN {X -21.4036,Y -111.5373,Z 115,A -104.1757,B 24.9537,C -1.5722,E1 24.9713,E2 190.096} C_DIS
LIN {X -15.6806,Y -112.4851,Z 115,A -100.4792,B 24.9517,C -1.605,E1 24.9817,E2 186.3186} C_DIS
LIN {X -10.7323,Y -113.0645,Z 115,A -98.9689,B 24.9544,C -1.5609,E1 24.9856,E2 184.912} C_DIS
LIN {X -5.6355,Y -113.4343,Z 115,A -96.0647,B 24.9535,C -1.5751,E1 24.9938,E2 181.9731} C_DIS
LIN {X -0.413,Y -113.572,Z 115,A -93.6682,B 24.9541,C -1.5651,E1 25.0004,E2 179.6} C_DIS
LIN {X -0.413,Y -113.572,Z 115,A -93.6682,B 24.9541,C -1.5651,E1 25.0004,E2 179.6} C_DIS
Enddeposition()
LIN {X 0.781,Y -112.6557,Z 115,A -92.9931,B 24.953,C -1.5843,E1 25.0024,E2 178.8795} C_DIS
Startdeposition()
$VEL.CP = VEL_PRINT
LIN {X -3.5557,Y -112.6033,Z 115,A -96.6034,B 24.9565,C -1.5239,E1 24.992,E2 182.6332} C_DIS
LIN {X -8.3057,Y -112.3547,Z 115,A -98.4477,B 24.9551,C -1.5481,E1 24.987,E2 184.4208} C_DIS
LIN {X -13.3697,Y -111.8632,Z 115,A -101.1569,B 24.9554,C -1.5433,E1 24.9794,E2 187.1431} C_DIS
LIN {X -18.4832,Y -111.1328,Z 115,A -103.5162,B 24.9547,C -1.5553,E1 24.973,E2 189.476} C_DIS
LIN {X -21.7901,Y -110.5331,Z 115,A -105.367,B 24.955,C -1.5499,E1 24.9679,E2 191.3415} C_DIS
LIN {X -25.3992,Y -109.7589,Z 115,A -107.1257,B 24.9546,C -1.5558,E1 24.9631,E2 193.0884} C_DIS
LIN {X -29.1416,Y -108.8253,Z 115,A -109.0797,B 24.9546,C -1.5573,E1 24.9578,E2 195.0417} C_DIS
LIN {X -32.5203,Y -107.8648,Z 115,A -111.1657,B 24.9552,C -1.546,E1 24.9522,E2 197.158} C_DIS
LIN {X -37.1636,Y -106.3533,Z 115,A -113.412,B 24.9545,C -1.5579,E1 24.9463,E2 199.3803} C_DIS
LIN {X -40.8662,Y -104.9867,Z 115,A -115.3995,B 24.9544,C -1.5606,E1 24.9411,E2 201.3655} C_DIS
LIN {X -45.0682,Y -103.2521,Z 115,A -117.7137,B 24.9542,C -1.563,E1 24.9351,E2 203.6795} C_DIS
LIN {X -48.5925,Y -101.6412,Z 115,A -119.6148,B 24.9539,C -1.5681,E1 24.9303,E2 205.573} C_DIS
LIN {X -51.346,Y -100.2782,Z 115,A -121.3008,B 24.9541,C -1.565,E1 24.9261,E2 207.271} C_DIS
LIN {X -54.9075,Y -98.3732,Z 115,A -123.2352,B 24.9537,C -1.5727,E1 24.9214,E2 209.1926} C_DIS
LIN {X -57.9311,Y -96.6259,Z 115,A -125.1424,B 24.9538,C -1.5699,E1 24.9168,E2 211.1123} C_DIS
LIN {X -61.2253,Y -94.5716,Z 115,A -126.9863,B 24.9533,C -1.5783,E1 24.9124,E2 212.9421} C_DIS
LIN {X -64.6282,Y -92.2793,Z 115,A -129.2352,B 24.9535,C -1.5751,E1 24.9072,E2 215.206} C_DIS
LIN {X -67.6726,Y -90.0697,Z 115,A -131.0701,B 24.9531,C -1.5816,E1 24.9031,E2 217.0319} C_DIS
LIN {X -70.3881,Y -87.9665,Z 115,A -132.9817,B 24.9533,C -1.5781,E1 24.8989,E2 218.959} C_DIS
LIN {X -73.4248,Y -85.4468,Z 115,A -134.939,B 24.953,C -1.584,E1 24.8947,E2 220.9099} C_DIS
LIN {X -76.3292,Y -82.8615,Z 115,A -136.9104,B 24.9527,C -1.5882,E1 24.8907,E2 222.8791} C_DIS
LIN {X -78.9655,Y -80.3533,Z 115,A -138.7517,B 24.9525,C -1.5925,E1 24.887,E2 224.7179} C_DIS
LIN {X -81.643,Y -77.6333,Z 115,A -140.5517,B 24.9519,C -1.6023,E1 24.8835,E2 226.5022} C_DIS
LIN {X -83.904,Y -75.1814,Z 115,A -142.7965,B 24.953,C -1.5843,E1 24.8792,E2 228.7998} C_DIS
LIN {X -86.2957,Y -72.4257,Z 115,A -144.2845,B 24.9518,C -1.6032,E1 24.8766,E2 230.2497} C_DIS
LIN {X -88.841,Y -69.2808,Z 115,A -146.5486,B 24.952,C -1.6,E1 24.8726,E2 232.5321} C_DIS
LIN {X -91.6477,Y -65.5198,Z 115,A -148.6637,B 24.951,C -1.6167,E1 24.8692,E2 234.6177} C_DIS
LIN {X -93.6697,Y -62.5979,Z 115,A -150.4261,B 24.9506,C -1.623,E1 24.8664,E2 236.3736} C_DIS
LIN {X -95.5206,Y -59.7322,Z 115,A -152.2818,B 24.9506,C -1.6228,E1 24.8636,E2 238.2392} C_DIS
LIN {X -97.4561,Y -56.5211,Z 115,A -154.326,B 24.9506,C -1.6225,E1 24.8607,E2 240.2947} C_DIS
LIN {X -98.8558,Y -54.0351,Z 115,A -156.0544,B 24.9511,C -1.6157,E1 24.8584,E2 242.0487} C_DIS
LIN {X -100.4884,Y -50.9347,Z 115,A -157.4134,B 24.9498,C -1.6372,E1 24.8567,E2 243.3636} C_DIS
LIN {X -101.9845,Y -47.8687,Z 115,A -159.2135,B 24.9496,C -1.6395,E1 24.8545,E2 245.1679} C_DIS
LIN {X -103.5718,Y -44.3329,Z 115,A -161.246,B 24.9494,C -1.6428,E1 24.8522,E2 247.2038} C_DIS
LIN {X -104.862,Y -41.1836,Z 115,A -162.9064,B 24.9489,C -1.6507,E1 24.8505,E2 248.8548} C_DIS
LIN {X -106.0377,Y -38.0589,Z 115,A -164.7409,B 24.9489,C -1.6503,E1 24.8487,E2 250.7003} C_DIS
LIN {X -107.3819,Y -34.0831,Z 115,A -166.9069,B 24.9486,C -1.6556,E1 24.8468,E2 252.8663} C_DIS
LIN {X -109.0106,Y -28.4425,Z 115,A -169.5585,B 24.9473,C -1.6777,E1 24.8449,E2 255.4804} C_DIS
LIN {X -109.9708,Y -24.4699,Z 115,A -171.8211,B 24.9473,C -1.677,E1 24.8434,E2 257.7581} C_DIS
LIN {X -110.493,Y -21.9973,Z 115,A -173.1792,B 24.9473,C -1.6782,E1 24.8426,E2 259.1214} C_DIS
LIN {X -110.9912,Y -19.3252,Z 115,A -174.7512,B 24.9474,C -1.6752,E1 24.8419,E2 260.7098} C_DIS
LIN {X -111.6912,Y -14.74,Z 115,A -176.9328,B 24.9465,C -1.6896,E1 24.841,E2 262.8701} C_DIS
LIN {X -112.119,Y -11.0428,Z 115,A -178.9485,B 24.9465,C -1.6909,E1 24.8404,E2 264.8947} C_DIS
LIN {X -112.4284,Y -7.2198,Z 115,A 179.2013,B 24.9458,C -1.7011,E1 24.84,E2 266.7318} C_DIS
LIN {X -112.6011,Y -3.6248,Z 115,A 177.3694,B 24.9454,C -1.7069,E1 24.8398,E2 268.5608} C_DIS
LIN {X -112.6594,Y -0.2798,Z 115,A 175.6932,B 24.945,C -1.7134,E1 24.8398,E2 270.2316} C_DIS
LIN {X -112.6123,Y 3.2598,Z 115,A 173.8999,B 24.9446,C -1.7195,E1 24.8398,E2 272.0211} C_DIS
LIN {X -112.4872,Y 6.2248,Z 115,A 172.3377,B 24.9444,C -1.7224,E1 24.8401,E2 273.5858} C_DIS
LIN {X -112.2211,Y 9.9362,Z 115,A 170.3627,B 24.9442,C -1.7254,E1 24.8405,E2 275.5657} C_DIS
LIN {X -111.813,Y 13.7999,Z 115,A 168.3092,B 24.944,C -1.7288,E1 24.8412,E2 277.6233} C_DIS
LIN {X -111.221,Y 17.9559,Z 115,A 165.7306,B 24.9446,C -1.7187,E1 24.8423,E2 280.2414} C_DIS
LIN {X -110.503,Y 21.9467,Z 115,A 164.0995,B 24.9431,C -1.7418,E1 24.8432,E2 281.8269} C_DIS
LIN {X -109.8219,Y 25.1265,Z 115,A 162.6191,B 24.9423,C -1.7539,E1 24.844,E2 283.2873} C_DIS
LIN {X -108.5193,Y 30.2638,Z 115,A 159.8968,B 24.9419,C -1.7614,E1 24.846,E2 286.0075} C_DIS
LIN {X -107.3973,Y 34.0291,Z 115,A 157.5665,B 24.9423,C -1.7549,E1 24.8479,E2 288.3667} C_DIS
LIN {X -106.0372,Y 38.0601,Z 115,A 155.5052,B 24.9416,C -1.7656,E1 24.8498,E2 290.4143} C_DIS
LIN {X -104.513,Y 42.0636,Z 115,A 152.7666,B 24.9425,C -1.7509,E1 24.8527,E2 293.2033} C_DIS
LIN {X -102.7347,Y 46.2355,Z 115,A 151.1861,B 24.9402,C -1.7858,E1 24.8544,E2 294.7091} C_DIS
LIN {X -101.4957,Y 48.8953,Z 115,A 149.6222,B 24.9402,C -1.7875,E1 24.8562,E2 296.2774} C_DIS
LIN {X -99.7742,Y 52.319,Z 115,A 147.7149,B 24.9396,C -1.795,E1 24.8586,E2 298.1772} C_DIS
LIN {X -97.9572,Y 55.6491,Z 115,A 144.9455,B 24.9414,C -1.7682,E1 24.8626,E2 301.025} C_DIS
LIN {X -95.428,Y 59.8805,Z 115,A 143.3436,B 24.9386,C -1.8103,E1 24.8648,E2 302.5346} C_DIS
LIN {X -92.3635,Y 64.5072,Z 115,A 140.3188,B 24.9386,C -1.8103,E1 24.8695,E2 305.5744} C_DIS
LIN {X -90.2324,Y 67.456,Z 115,A 137.9737,B 24.9395,C -1.7962,E1 24.8735,E2 307.9645} C_DIS
LIN {X -87.8198,Y 70.5694,Z 115,A 136.2708,B 24.9384,C -1.8131,E1 24.8764,E2 309.6351} C_DIS
LIN {X -85.0928,Y 73.834,Z 115,A 134.2672,B 24.9376,C -1.825,E1 24.88,E2 311.6196} C_DIS
LIN {X -82.8293,Y 76.3643,Z 115,A 132.5959,B 24.9371,C -1.8316,E1 24.8831,E2 313.2827} C_DIS
LIN {X -79.9761,Y 79.3475,Z 115,A 130.2973,B 24.9373,C -1.8289,E1 24.8876,E2 315.5974} C_DIS
LIN {X -77.1736,Y 82.0753,Z 115,A 128.4665,B 24.9365,C -1.8399,E1 24.8912,E2 317.4097} C_DIS
LIN {X -74.6795,Y 84.3534,Z 115,A 126.6452,B 24.9365,C -1.8398,E1 24.895,E2 319.2386} C_DIS
LIN {X -72.5897,Y 86.1583,Z 115,A 125.1626,B 24.9365,C -1.8398,E1 24.8982,E2 320.7267} C_DIS
LIN {X -68.5105,Y 89.4346,Z 115,A 122.6437,B 24.9358,C -1.8512,E1 24.9037,E2 323.2279} C_DIS
LIN {X -65.5579,Y 91.6205,Z 115,A 120.7701,B 24.9355,C -1.8549,E1 24.9079,E2 325.0993} C_DIS
LIN {X -62.9252,Y 93.4485,Z 115,A 119.1098,B 24.9354,C -1.8569,E1 24.9117,E2 326.7603} C_DIS
LIN {X -59.4321,Y 95.7081,Z 115,A 116.8871,B 24.9354,C -1.8567,E1 24.917,E2 328.9906} C_DIS
LIN {X -56.8141,Y 97.2863,Z 115,A 115.348,B 24.9351,C -1.8601,E1 24.9207,E2 330.5263} C_DIS
LIN {X -51.3651,Y 100.2684,Z 115,A 112.0734,B 24.9351,C -1.8609,E1 24.9288,E2 333.8082} C_DIS
LIN {X -47.5192,Y 102.1472,Z 115,A 110.0556,B 24.9344,C -1.8707,E1 24.9338,E2 335.8078} C_DIS
LIN {X -45.3013,Y 103.1504,Z 115,A 108.1552,B 24.9361,C -1.846,E1 24.9389,E2 337.7714} C_DIS
LIN {X -41.0152,Y 104.9281,Z 115,A 106.5055,B 24.9339,C -1.8778,E1 24.9429,E2 339.3492} C_DIS
LIN {X -37.9112,Y 106.0909,Z 115,A 104.7349,B 24.9339,C -1.8765,E1 24.9476,E2 341.1265} C_DIS
LIN {X -31.7552,Y 108.0917,Z 115,A 101.5246,B 24.9335,C -1.8837,E1 24.9561,E2 344.3255} C_DIS
LIN {X -27.3895,Y 109.2813,Z 115,A 99.1142,B 24.9336,C -1.8815,E1 24.9626,E2 346.7445} C_DIS
LIN {X -24.2205,Y 110.0252,Z 115,A 97.5557,B 24.9332,C -1.887,E1 24.9669,E2 348.292} C_DIS
LIN {X -21.4022,Y 110.6078,Z 115,A 96.0894,B 24.9332,C -1.8881,E1 24.9709,E2 349.7573} C_DIS
LIN {X -17.9443,Y 111.2229,Z 115,A 94.1822,B 24.9334,C -1.8845,E1 24.9761,E2 351.6751} C_DIS
LIN {X -14.5904,Y 111.7106,Z 115,A 92.5521,B 24.9331,C -1.8894,E1 24.9806,E2 353.2946} C_DIS
LIN {X -9.2375,Y 112.2803,Z 115,A 89.6186,B 24.9335,C -1.8828,E1 24.9888,E2 356.2456} C_DIS
LIN {X -5.0888,Y 112.5446,Z 115,A 86.936,B 24.9351,C -1.8601,E1 24.9965,E2 358.9825} C_DIS
LIN {X -0.1328,Y 112.6606,Z 115,A 84.9743,B 24.9335,C -1.8837,E1 25.0018,E2 360.8882} C_DIS
LIN {X 5.0841,Y 112.5448,Z 115,A 82.4796,B 24.933,C -1.8906,E1 25.0087,E2 363.3661} C_DIS
LIN {X 8.9018,Y 112.3071,Z 115,A 80.5603,B 24.933,C -1.8917,E1 25.014,E2 365.282} C_DIS
LIN {X 11.9521,Y 112.0238,Z 115,A 79.081,B 24.9327,C -1.8948,E1 25.0181,E2 366.753} C_DIS
LIN {X 15.3396,Y 111.6113,Z 115,A 77.2889,B 24.9329,C -1.892,E1 25.0231,E2 368.5503} C_DIS
LIN {X 18.4763,Y 111.134,Z 115,A 75.6277,B 24.9331,C -1.8895,E1 25.0277,E2 370.2158} C_DIS
LIN {X 22.2272,Y 110.4458,Z 115,A 73.6607,B 24.9332,C -1.8875,E1 25.0331,E2 372.1852} C_DIS
LIN {X 25.6057,Y 109.7112,Z 115,A 71.9821,B 24.933,C -1.89,E1 25.0376,E2 373.8556} C_DIS
LIN {X 29.6186,Y 108.6965,Z 115,A 69.5185,B 24.9342,C -1.8734,E1 25.0444,E2 376.3547} C_DIS
LIN {X 32.7541,Y 107.7947,Z 115,A 68.0443,B 24.9337,C -1.88,E1 25.0483,E2 377.8107} C_DIS
LIN {X 36.7505,Y 106.4982,Z 115,A 66.0796,B 24.9334,C -1.8856,E1 25.0534,E2 379.7584} C_DIS
LIN {X 39.6642,Y 105.4464,Z 115,A 64.2567,B 24.9342,C -1.8735,E1 25.0583,E2 381.606} C_DIS
LIN {X 43.8046,Y 103.7944,Z 115,A 62.2533,B 24.9336,C -1.8825,E1 25.0634,E2 383.5836} C_DIS
LIN {X 46.0193,Y 102.8321,Z 115,A 60.7736,B 24.9344,C -1.8702,E1 25.0672,E2 385.0886} C_DIS
LIN {X 51.3202,Y 100.2914,Z 115,A 58.0294,B 24.934,C -1.8771,E1 25.0741,E2 387.8093} C_DIS
LIN {X 54.8137,Y 98.4256,Z 115,A 56.0674,B 24.934,C -1.8766,E1 25.0789,E2 389.7668} C_DIS
LIN {X 57.5805,Y 96.8334,Z 115,A 54.3021,B 24.9346,C -1.868,E1 25.0831,E2 391.547} C_DIS
LIN {X 60.7067,Y 94.9044,Z 115,A 52.5555,B 24.9344,C -1.8704,E1 25.0873,E2 393.2823} C_DIS
LIN {X 63.1481,Y 93.2976,Z 115,A 51.1965,B 24.9342,C -1.8736,E1 25.0904,E2 394.6294} C_DIS
LIN {X 65.038,Y 91.9914,Z 115,A 49.8513,B 24.9349,C -1.8638,E1 25.0935,E2 395.9929} C_DIS
LIN {X 67.8594,Y 89.9293,Z 115,A 48.0592,B 24.9351,C -1.86,E1 25.0975,E2 397.7876} C_DIS
LIN {X 70.2051,Y 88.1111,Z 115,A 46.2886,B 24.9361,C -1.8457,E1 25.1015,E2 399.5853} C_DIS
LIN {X 73.8255,Y 85.1004,Z 115,A 44.2058,B 24.9355,C -1.8548,E1 25.1058,E2 401.6387} C_DIS
LIN {X 75.9833,Y 83.1789,Z 115,A 42.1327,B 24.9376,C -1.8253,E1 25.1102,E2 403.7731} C_DIS
LIN {X 79.2043,Y 80.1174,Z 115,A 40.9301,B 24.9346,C -1.8671,E1 25.1125,E2 404.8718} C_DIS
LIN {X 83.939,Y 75.1423,Z 115,A 37.0411,B 24.9364,C -1.8417,E1 25.12,E2 408.804} C_DIS
LIN {X 86.1528,Y 72.5961,Z 115,A 35.1324,B 24.9373,C -1.829,E1 25.1235,E2 410.7338} C_DIS
LIN {X 90.0975,Y 67.6356,Z 115,A 32.1406,B 24.9371,C -1.8315,E1 25.1286,E2 413.7056} C_DIS
LIN {X 92.3037,Y 64.5932,Z 115,A 30.1468,B 24.9377,C -1.823,E1 25.1318,E2 415.7099} C_DIS
LIN {X 94.6095,Y 61.1663,Z 115,A 28.3341,B 24.9372,C -1.8305,E1 25.1346,E2 417.4959} C_DIS
LIN {X 96.3166,Y 58.4401,Z 115,A 26.5087,B 24.9381,C -1.8176,E1 25.1373,E2 419.3424} C_DIS
LIN {X 98.1592,Y 55.2908,Z 115,A 24.5132,B 24.9388,C -1.8063,E1 25.1401,E2 421.3544} C_DIS
LIN {X 100.2141,Y 51.4715,Z 115,A 22.4384,B 24.9388,C -1.8061,E1 25.1428,E2 423.4187} C_DIS
LIN {X 101.8957,Y 48.0596,Z 115,A 20.5295,B 24.9392,C -1.8017,E1 25.1451,E2 425.3277} C_DIS
LIN {X 103.3008,Y 44.9565,Z 115,A 18.2207,B 24.9412,C -1.7708,E1 25.1478,E2 427.6967} C_DIS
LIN {X 104.964,Y 40.924,Z 115,A 16.0026,B 24.9417,C -1.7643,E1 25.15,E2 429.9179} C_DIS
LIN {X 106.5052,Y 36.7306,Z 115,A 14.3149,B 24.9404,C -1.7838,E1 25.1515,E2 431.5502} C_DIS
LIN {X 107.5237,Y 33.6282,Z 115,A 12.4419,B 24.9413,C -1.7691,E1 25.1531,E2 433.4471} C_DIS
LIN {X 108.7125,Y 29.5593,Z 115,A 10.6659,B 24.9406,C -1.7797,E1 25.1544,E2 435.1879} C_DIS
LIN {X 109.5031,Y 26.4812,Z 115,A 8.9302,B 24.9413,C -1.7693,E1 25.1556,E2 436.9382} C_DIS
LIN {X 110.2995,Y 22.9397,Z 115,A 7.1122,B 24.9416,C -1.7648,E1 25.1567,E2 438.7562} C_DIS
LIN {X 110.9437,Y 19.5895,Z 115,A 5.4194,B 24.9419,C -1.7612,E1 25.1576,E2 440.4476} C_DIS
LIN {X 111.5269,Y 15.9341,Z 115,A 3.5917,B 24.9421,C -1.7577,E1 25.1583,E2 442.2726} C_DIS
LIN {X 111.8825,Y 13.2078,Z 115,A 2.1443,B 24.9425,C -1.751,E1 25.1588,E2 443.7273} C_DIS
LIN {X 112.2712,Y 9.3515,Z 115,A 0.2187,B 24.9428,C -1.7468,E1 25.1593,E2 445.6516} C_DIS
LIN {X 112.6301,Y 2.6233,Z 115,A -3.0699,B 24.9431,C -1.7419,E1 25.1598,E2 448.932} C_DIS
LIN {X 112.6104,Y -3.3228,Z 115,A -5.889,B 24.9431,C -1.7415,E1 25.1598,E2 451.7355} C_DIS
LIN {X 112.5105,Y -5.804,Z 115,A -8.0339,B 24.946,C -1.6971,E1 25.1594,E2 453.9722} C_DIS
LIN {X 112.2181,Y -9.9686,Z 115,A -9.7403,B 24.9453,C -1.7091,E1 25.159,E2 455.6402} C_DIS
LIN {X 111.7377,Y -14.381,Z 115,A -11.752,B 24.945,C -1.713,E1 25.1584,E2 457.6309} C_DIS
LIN {X 111.3051,Y -17.4171,Z 115,A -13.4045,B 24.9456,C -1.7037,E1 25.1577,E2 459.2956} C_DIS
LIN {X 110.667,Y -21.0945,Z 115,A -15.2304,B 24.9458,C -1.7008,E1 25.1568,E2 461.1174} C_DIS
LIN {X 109.9662,Y -24.4909,Z 115,A -17.0995,B 24.9465,C -1.6903,E1 25.1557,E2 463.0005} C_DIS
LIN {X 109.1468,Y -27.9127,Z 115,A -18.7576,B 24.9465,C -1.6906,E1 25.1546,E2 464.6484} C_DIS
LIN {X 107.9789,Y -32.1356,Z 115,A -20.9391,B 24.9468,C -1.6856,E1 25.1529,E2 466.8292} C_DIS
LIN {X 106.9968,Y -35.2731,Z 115,A -22.6552,B 24.9472,C -1.6783,E1 25.1514,E2 468.5528} C_DIS
LIN {X 105.7291,Y -38.9048,Z 115,A -24.5908,B 24.9475,C -1.6731,E1 25.1496,E2 470.4897} C_DIS
LIN {X 104.3883,Y -42.37,Z 115,A -26.5719,B 24.9482,C -1.6631,E1 25.1476,E2 472.4834} C_DIS
LIN {X 102.748,Y -46.2058,Z 115,A -28.461,B 24.9479,C -1.6672,E1 25.1455,E2 474.3526} C_DIS
LIN {X 100.4651,Y -50.9803,Z 115,A -31.3368,B 24.9489,C -1.6506,E1 25.1419,E2 477.252} C_DIS
LIN {X 98.5302,Y -54.6264,Z 115,A -33.3495,B 24.9491,C -1.6483,E1 25.1393,E2 479.2595} C_DIS
LIN {X 96.9784,Y -57.3351,Z 115,A -34.9172,B 24.9493,C -1.6446,E1 25.1371,E2 480.828} C_DIS
LIN {X 95.6742,Y -59.4864,Z 115,A -36.3177,B 24.9499,C -1.6354,E1 25.135,E2 482.2431} C_DIS
LIN {X 92.7268,Y -63.9845,Z 115,A -38.971,B 24.9501,C -1.6314,E1 25.1309,E2 484.8927} C_DIS
LIN {X 90.4924,Y -67.1098,Z 115,A -40.9271,B 24.9505,C -1.6258,E1 25.1276,E2 486.8524} C_DIS
LIN {X 88.439,Y -69.7902,Z 115,A -42.5536,B 24.9505,C -1.6253,E1 25.1249,E2 488.4725} C_DIS
LIN {X 86.0652,Y -72.699,Z 115,A -44.514,B 24.9509,C -1.618,E1 25.1214,E2 490.4412} C_DIS
LIN {X 83.6933,Y -75.4167,Z 115,A -46.2763,B 24.951,C -1.6165,E1 25.1181,E2 492.1991} C_DIS
LIN {X 81.1973,Y -78.097,Z 115,A -48.096,B 24.9512,C -1.6137,E1 25.1146,E2 494.0174} C_DIS
LIN {X 78.9934,Y -80.3258,Z 115,A -49.687,B 24.9514,C -1.61,E1 25.1115,E2 495.6106} C_DIS
LIN {X 76.2722,Y -82.9138,Z 115,A -51.5977,B 24.9517,C -1.6054,E1 25.1076,E2 497.5243} C_DIS
LIN {X 73.6655,Y -85.2401,Z 115,A -53.4681,B 24.9522,C -1.597,E1 25.1036,E2 499.407} C_DIS
LIN {X 70.8432,Y -87.5979,Z 115,A -55.2366,B 24.9522,C -1.5974,E1 25.0998,E2 501.1678} C_DIS
LIN {X 67.8326,Y -89.9495,Z 115,A -57.1664,B 24.9524,C -1.5938,E1 25.0955,E2 503.0992} C_DIS
LIN {X 65.0907,Y -91.9538,Z 115,A -58.9934,B 24.9529,C -1.5857,E1 25.0914,E2 504.9388} C_DIS
LIN {X 61.6236,Y -94.3127,Z 115,A -61.6186,B 24.9544,C -1.5596,E1 25.0851,E2 507.6169} C_DIS
LIN {X 57.9668,Y -96.6043,Z 115,A -63.3109,B 24.9534,C -1.5777,E1 25.0812,E2 509.2612} C_DIS
LIN {X 54.9799,Y -98.3328,Z 115,A -64.9228,B 24.9532,C -1.5809,E1 25.0773,E2 510.8607} C_DIS
LIN {X 52.3139,Y -99.7769,Z 115,A -66.566,B 24.9536,C -1.5738,E1 25.0732,E2 512.5162} C_DIS
LIN {X 47.866,Y -101.9858,Z 115,A -68.9969,B 24.9536,C -1.5738,E1 25.0672,E2 514.9405} C_DIS
LIN {X 42.5803,Y -104.3027,Z 115,A -72.2343,B 24.9546,C -1.5562,E1 25.0588,E2 518.2119} C_DIS
LIN {X 36.5808,Y -106.5568,Z 115,A -75.2488,B 24.9543,C -1.5625,E1 25.0509,E2 521.2051} C_DIS
LIN {X 33.9243,Y -107.4319,Z 115,A -76.6769,B 24.9543,C -1.5606,E1 25.0471,E2 522.6352} C_DIS
LIN {X 30.5215,Y -108.4463,Z 115,A -78.4633,B 24.9544,C -1.5594,E1 25.0423,E2 524.4213} C_DIS
LIN {X 26.7864,Y -109.4286,Z 115,A -80.3203,B 24.9543,C -1.5621,E1 25.0373,E2 526.2693} C_DIS
LIN {X 23.5882,Y -110.1631,Z 115,A -82.068,B 24.9546,C -1.5571,E1 25.0325,E2 528.0265} C_DIS
LIN {X 20.7227,Y -110.7386,Z 115,A -83.8018,B 24.9553,C -1.5451,E1 25.0277,E2 529.7866} C_DIS
LIN {X 15.4564,Y -111.5947,Z 115,A -86.318,B 24.9549,C -1.5517,E1 25.0208,E2 532.2849} C_DIS
LIN {X 8.776,Y -112.3172,Z 115,A -90.3534,B 24.9565,C -1.5234,E1 25.0094,E2 536.3847} C_DIS
LIN {X 3.9932,Y -112.589,Z 115,A -92.059,B 24.9548,C -1.5537,E1 25.0048,E2 538.0182} C_DIS
LIN {X 0.781,Y -112.6557,Z 115,A -92.9911,B 24.953,C -1.5835,E1 25.0025,E2 538.8795} C_DIS
Enddeposition()
LIN {X 0.781,Y -112.6557,Z 115,A -92.9911,B 24.953,C -1.5835,E1 25.0025,E2 538.8795} C_DIS
Startdeposition()
$VEL.CP = VEL_PRINT
LIN {X 2.3515,Y -111.7219,Z 115,A -92.0685,B 24.9518,C -1.6045,E1 25.0052,E2 537.9071} C_DIS
LIN {X 9.5735,Y -111.3364,Z 115,A -88.0089,B 24.9507,C -1.6214,E1 25.0166,E2 533.8094} C_DIS
LIN {X 13.0667,Y -110.9797,Z 115,A -87.0728,B 24.9529,C -1.5849,E1 25.0189,E2 532.9602} C_DIS
LIN {X 15.4652,Y -110.6713,Z 115,A -85.395,B 24.9517,C -1.6047,E1 25.0237,E2 531.237} C_DIS
LIN {X 20.9391,Y -109.7671,Z 115,A -82.4842,B 24.9514,C -1.6098,E1 25.0317,E2 528.3173} C_DIS
LIN {X 24.8202,Y -108.9555,Z 115,A -80.5234,B 24.9515,C -1.6085,E1 25.0371,E2 526.3621} C_DIS
LIN {X 27.8731,Y -108.2143,Z 115,A -78.9267,B 24.9515,C -1.6095,E1 25.0414,E2 524.7654} C_DIS
LIN {X 31.9282,Y -107.0881,Z 115,A -76.8754,B 24.9515,C -1.6073,E1 25.0469,E2 522.7229} C_DIS
LIN {X 34.5593,Y -106.2681,Z 115,A -75.3891,B 24.9513,C -1.6122,E1 25.0508,E2 521.2277} C_DIS
LIN {X 40.5612,Y -104.1255,Z 115,A -72.3573,B 24.9517,C -1.6061,E1 25.0588,E2 518.2166} C_DIS
LIN {X 45.2799,Y -102.1637,Z 115,A -69.5787,B 24.951,C -1.6169,E1 25.066,E2 515.4191} C_DIS
LIN {X 48.6478,Y -100.6017,Z 115,A -67.4477,B 24.9502,C -1.6301,E1 25.0714,E2 513.2623} C_DIS
LIN {X 52.3703,Y -98.7153,Z 115,A -65.617,B 24.9508,C -1.6199,E1 25.0759,E2 511.4607} C_DIS
LIN {X 54.5572,Y -97.5231,Z 115,A -64.1879,B 24.9503,C -1.629,E1 25.0794,E2 510.0143} C_DIS
LIN {X 61.9038,Y -93.0343,Z 115,A -59.8227,B 24.9499,C -1.6351,E1 25.0898,E2 505.6486} C_DIS
LIN {X 64.6729,Y -91.1303,Z 115,A -58.1073,B 24.9497,C -1.6383,E1 25.0937,E2 503.9316} C_DIS
LIN {X 67.1872,Y -89.2924,Z 115,A -56.4863,B 24.9494,C -1.6428,E1 25.0973,E2 502.3057} C_DIS
LIN {X 70.2909,Y -86.8702,Z 115,A -54.497,B 24.9492,C -1.6459,E1 25.1017,E2 500.3165} C_DIS
LIN {X 73.0416,Y -84.5727,Z 115,A -52.4985,B 24.9485,C -1.6573,E1 25.106,E2 498.2987} C_DIS
LIN {X 76.1455,Y -81.7889,Z 115,A -50.4626,B 24.9485,C -1.6578,E1 25.1101,E2 496.2701} C_DIS
LIN {X 78.5431,Y -79.4872,Z 115,A -48.8546,B 24.9485,C -1.6576,E1 25.1133,E2 494.6692} C_DIS
LIN {X 80.8992,Y -77.0906,Z 115,A -47.0088,B 24.9479,C -1.6674,E1 25.1169,E2 492.8081} C_DIS
LIN {X 83.4921,Y -74.2727,Z 115,A -45.2176,B 24.9481,C -1.6647,E1 25.1203,E2 491.0315} C_DIS
LIN {X 85.5319,Y -71.9162,Z 115,A -43.4786,B 24.9474,C -1.6752,E1 25.1235,E2 489.2754} C_DIS
LIN {X 87.7304,Y -69.2143,Z 115,A -41.8066,B 24.9474,C -1.6749,E1 25.1264,E2 487.612} C_DIS
LIN {X 89.7992,Y -66.5111,Z 115,A -40.0884,B 24.9472,C -1.6784,E1 25.1292,E2 485.8938} C_DIS
LIN {X 91.8266,Y -63.6799,Z 115,A -37.6535,B 24.945,C -1.7132,E1 25.1332,E2 483.3887} C_DIS
LIN {X 94.3274,Y -59.9154,Z 115,A -35.4896,B 24.945,C -1.7127,E1 25.1365,E2 481.2368} C_DIS
LIN {X 96.3066,Y -56.6774,Z 115,A -34.1227,B 24.9464,C -1.6918,E1 25.1383,E2 479.9262} C_DIS
LIN {X 97.9795,Y -53.7357,Z 115,A -31.0125,B 24.9419,C -1.7606,E1 25.1427,E2 476.6701} C_DIS
LIN {X 101.3063,Y -47.1621,Z 115,A -28.6636,B 24.9455,C -1.7057,E1 25.1454,E2 474.4632} C_DIS
LIN {X 102.6504,Y -44.1636,Z 115,A -26.8216,B 24.9447,C -1.7181,E1 25.1474,E2 472.6021} C_DIS
LIN {X 104.2882,Y -40.1445,Z 115,A -24.7965,B 24.9448,C -1.7158,E1 25.1495,E2 470.5936} C_DIS
LIN {X 105.4422,Y -37.0025,Z 115,A -23.0103,B 24.9443,C -1.7244,E1 25.1512,E2 468.7971} C_DIS
LIN {X 106.6127,Y -33.4834,Z 115,A -20.561,B 24.9422,C -1.7557,E1 25.1533,E2 466.2879} C_DIS
LIN {X 107.754,Y -29.6064,Z 115,A -19.1899,B 24.9439,C -1.7299,E1 25.1543,E2 464.9854} C_DIS
LIN {X 108.5182,Y -26.666,Z 115,A -17.5144,B 24.9432,C -1.7404,E1 25.1555,E2 463.2951} C_DIS
LIN {X 109.2445,Y -23.5151,Z 115,A -15.8998,B 24.943,C -1.7437,E1 25.1565,E2 461.6819} C_DIS
LIN {X 109.9598,Y -19.9023,Z 115,A -13.9649,B 24.9425,C -1.752,E1 25.1575,E2 459.7388} C_DIS
LIN {X 110.5625,Y -16.2309,Z 115,A -11.9694,B 24.9418,C -1.7622,E1 25.1583,E2 457.731} C_DIS
LIN {X 111.0436,Y -12.5212,Z 115,A -10.2367,B 24.942,C -1.7599,E1 25.1589,E2 456.0139} C_DIS
LIN {X 111.63,Y -5.1061,Z 115,A -6.5845,B 24.9416,C -1.7648,E1 25.1597,E2 452.3718} C_DIS
LIN {X 111.7276,Y -2.0432,Z 115,A -4.2569,B 24.9389,C -1.8048,E1 25.1597,E2 449.9637} C_DIS
LIN {X 111.7264,Y 2.1102,Z 115,A -2.9278,B 24.941,C -1.7748,E1 25.1597,E2 448.7133} C_DIS
LIN {X 111.5619,Y 6.4213,Z 115,A -0.5807,B 24.9401,C -1.7881,E1 25.1595,E2 446.3488} C_DIS
LIN {X 111.3059,Y 9.9179,Z 115,A 1.5825,B 24.9385,C -1.8108,E1 25.1589,E2 444.145} C_DIS
LIN {X 110.8526,Y 14.1067,Z 115,A 3.3887,B 24.9392,C -1.8014,E1 25.1584,E2 442.3716} C_DIS
LIN {X 110.4218,Y 17.1544,Z 115,A 4.9962,B 24.9387,C -1.8077,E1 25.1577,E2 440.7586} C_DIS
LIN {X 109.797,Y 20.7841,Z 115,A 6.887,B 24.9383,C -1.8138,E1 25.1568,E2 438.8646} C_DIS
LIN {X 109.0802,Y 24.2684,Z 115,A 8.7616,B 24.9378,C -1.8218,E1 25.1556,E2 436.9819} C_DIS
LIN {X 108.2243,Y 27.8343,Z 115,A 10.4575,B 24.938,C -1.8193,E1 25.1545,E2 435.3019} C_DIS
LIN {X 107.405,Y 30.8474,Z 115,A 12.6592,B 24.9357,C -1.8517,E1 25.1528,E2 433.0363} C_DIS
LIN {X 106.2467,Y 34.6255,Z 115,A 14.0517,B 24.9373,C -1.8288,E1 25.1517,E2 431.7056} C_DIS
LIN {X 105.0493,Y 38.104,Z 115,A 16.3787,B 24.9355,C -1.8546,E1 25.1494,E2 429.3309} C_DIS
LIN {X 103.8886,Y 41.1643,Z 115,A 18.0279,B 24.9353,C -1.8582,E1 25.1477,E2 427.6824} C_DIS
LIN {X 102.6558,Y 44.1512,Z 115,A 19.1956,B 24.9365,C -1.8407,E1 25.1465,E2 426.5623} C_DIS
LIN {X 100.7958,Y 48.2439,Z 115,A 21.6015,B 24.9357,C -1.8519,E1 25.1437,E2 424.143} C_DIS
LIN {X 99.2381,Y 51.375,Z 115,A 23.4881,B 24.9351,C -1.8611,E1 25.1413,E2 422.2446} C_DIS
LIN {X 97.0037,Y 55.4759,Z 115,A 25.8088,B 24.9348,C -1.8644,E1 25.1381,E2 419.9284} C_DIS
LIN {X 94.6041,Y 59.476,Z 115,A 27.9405,B 24.9352,C -1.859,E1 25.1351,E2 417.8202} C_DIS
LIN {X 93.2017,Y 61.6498,Z 115,A 29.4294,B 24.9345,C -1.8698,E1 25.1328,E2 416.3133} C_DIS
LIN {X 91.1928,Y 64.5853,Z 115,A 31.2764,B 24.9341,C -1.8755,E1 25.1298,E2 414.462} C_DIS
LIN {X 89.3985,Y 67.0459,Z 115,A 33.1312,B 24.9329,C -1.8926,E1 25.1267,E2 412.5757} C_DIS
LIN {X 86.5905,Y 70.6361,Z 115,A 35.3442,B 24.9329,C -1.8926,E1 25.1228,E2 410.373} C_DIS
LIN {X 84.0509,Y 73.639,Z 115,A 37.1656,B 24.9331,C -1.8886,E1 25.1195,E2 408.5694} C_DIS
LIN {X 79.2517,Y 78.7815,Z 115,A 40.8294,B 24.9324,C -1.899,E1 25.1125,E2 404.8967} C_DIS
LIN {X 75.0842,Y 82.7647,Z 115,A 43.6297,B 24.9324,C -1.8982,E1 25.1068,E2 402.1098} C_DIS
LIN {X 71.8366,Y 85.5981,Z 115,A 46.1582,B 24.9311,C -1.9167,E1 25.1014,E2 399.5475} C_DIS
LIN {X 68.9301,Y 87.955,Z 115,A 47.9727,B 24.9312,C -1.9156,E1 25.0974,E2 397.7422} C_DIS
LIN {X 65.7711,Y 90.341,Z 115,A 49.9761,B 24.931,C -1.9181,E1 25.0929,E2 395.7403} C_DIS
LIN {X 62.5374,Y 92.6085,Z 115,A 51.6709,B 24.9318,C -1.907,E1 25.0891,E2 394.0776} C_DIS
LIN {X 60.2473,Y 94.1144,Z 115,A 53.2171,B 24.9312,C -1.9154,E1 25.0855,E2 392.5165} C_DIS
LIN {X 57.8163,Y 95.6273,Z 115,A 54.826,B 24.9306,C -1.9238,E1 25.0816,E2 390.8928} C_DIS
LIN {X 54.9029,Y 97.33,Z 115,A 56.6257,B 24.9302,C -1.9293,E1 25.0772,E2 389.0854} C_DIS
LIN {X 51.7591,Y 99.0371,Z 115,A 58.2282,B 24.9308,C -1.9217,E1 25.0733,E2 387.5056} C_DIS
LIN {X 46.4595,Y 101.6322,Z 115,A 61.1891,B 24.9308,C -1.9225,E1 25.0659,E2 384.5503} C_DIS
LIN {X 44.0707,Y 102.6909,Z 115,A 62.7495,B 24.9299,C -1.9336,E1 25.0618,E2 382.9676} C_DIS
LIN {X 40.6468,Y 104.0919,Z 115,A 64.6522,B 24.9297,C -1.9358,E1 25.0569,E2 381.0639} C_DIS
LIN {X 36.4923,Y 105.6212,Z 115,A 66.7034,B 24.9303,C -1.9284,E1 25.0515,E2 379.0345} C_DIS
LIN {X 33.5125,Y 106.6036,Z 115,A 69.0739,B 24.9278,C -1.9626,E1 25.045,E2 376.5873} C_DIS
LIN {X 29.1602,Y 107.8745,Z 115,A 70.6871,B 24.9299,C -1.9335,E1 25.0409,E2 375.0457} C_DIS
LIN {X 26.02,Y 108.6758,Z 115,A 72.3114,B 24.9299,C -1.9328,E1 25.0365,E2 373.4253} C_DIS
LIN {X 22.8941,Y 109.3768,Z 115,A 74.054,B 24.9296,C -1.9379,E1 25.0317,E2 371.6729} C_DIS
LIN {X 19.1708,Y 110.0913,Z 115,A 76.0817,B 24.9293,C -1.9422,E1 25.0261,E2 369.6373} C_DIS
LIN {X 15.6789,Y 110.6409,Z 115,A 77.7692,B 24.9296,C -1.9375,E1 25.0215,E2 367.9626} C_DIS
LIN {X 11.5534,Y 111.1475,Z 115,A 79.9534,B 24.9294,C -1.9401,E1 25.0154,E2 365.7738} C_DIS
LIN {X 7.0187,Y 111.5269,Z 115,A 82.2291,B 24.9296,C -1.9377,E1 25.0091,E2 363.5047} C_DIS
LIN {X 3.5184,Y 111.6909,Z 115,A 84.3749,B 24.9285,C -1.9523,E1 25.003,E2 361.3249} C_DIS
LIN {X -0.6815,Y 111.7442,Z 115,A 86.6817,B 24.9281,C -1.9583,E1 24.9965,E2 359.0039} C_DIS
LIN {X -4.4896,Y 111.6565,Z 115,A 87.8978,B 24.9304,C -1.9269,E1 24.9934,E2 357.8623} C_DIS
LIN {X -8.6264,Y 111.4132,Z 115,A 90.9181,B 24.9277,C -1.9634,E1 24.9847,E2 354.7542} C_DIS
LIN {X -13.0374,Y 110.9832,Z 115,A 92.5587,B 24.9298,C -1.9357,E1 24.9803,E2 353.1782} C_DIS
LIN {X -16.892,Y 110.4623,Z 115,A 94.5415,B 24.9298,C -1.9339,E1 24.9748,E2 351.198} C_DIS
LIN {X -20.3852,Y 109.8729,Z 115,A 96.4709,B 24.9296,C -1.9372,E1 24.9695,E2 349.2588} C_DIS
LIN {X -23.7707,Y 109.1888,Z 115,A 98.1041,B 24.9302,C -1.93,E1 24.9651,E2 347.6407} C_DIS
LIN {X -27.139,Y 108.4028,Z 115,A 100.4171,B 24.9287,C -1.9505,E1 24.9587,E2 345.2758} C_DIS
LIN {X -30.7401,Y 107.4354,Z 115,A 101.7128,B 24.9307,C -1.9232,E1 24.9554,E2 344.043} C_DIS
LIN {X -37.8883,Y 105.128,Z 115,A 105.5016,B 24.9312,C -1.9159,E1 24.9454,E2 340.2646} C_DIS
LIN {X -45.3985,Y 102.1104,Z 115,A 109.7274,B 24.9314,C -1.913,E1 24.9344,E2 336.0363} C_DIS
LIN {X -48.1784,Y 100.8272,Z 115,A 111.4099,B 24.9312,C -1.9151,E1 24.9301,E2 334.3445} C_DIS
LIN {X -55.2095,Y 97.1567,Z 115,A 115.4269,B 24.9319,C -1.9061,E1 24.9203,E2 330.3377} C_DIS
LIN {X -57.8503,Y 95.6066,Z 115,A 117.1061,B 24.9318,C -1.9076,E1 24.9162,E2 328.6498} C_DIS
LIN {X -61.9986,Y 92.9718,Z 115,A 119.515,B 24.9324,C -1.8983,E1 24.9106,E2 326.2553} C_DIS
LIN {X -64.646,Y 91.1495,Z 115,A 121.3137,B 24.9323,C -1.901,E1 24.9064,E2 324.444} C_DIS
LIN {X -67.2435,Y 89.25,Z 115,A 123.5602,B 24.9308,C -1.9215,E1 24.9013,E2 322.1407} C_DIS
LIN {X -70.6954,Y 86.5423,Z 115,A 125.5782,B 24.9318,C -1.9072,E1 24.897,E2 320.149} C_DIS
LIN {X -73.2218,Y 84.4153,Z 115,A 126.959,B 24.933,C -1.8909,E1 24.8941,E2 318.8017} C_DIS
LIN {X -75.8157,Y 82.0935,Z 115,A 128.6521,B 24.9335,C -1.8831,E1 24.8907,E2 317.1203} C_DIS
LIN {X -79.5618,Y 78.4676,Z 115,A 131.8434,B 24.9325,C -1.8972,E1 24.8842,E2 313.8821} C_DIS
LIN {X -82.1115,Y 75.7961,Z 115,A 133.0441,B 24.9348,C -1.8651,E1 24.8821,E2 312.7527} C_DIS
LIN {X -83.9047,Y 73.8065,Z 115,A 134.6709,B 24.9343,C -1.8715,E1 24.879,E2 311.1033} C_DIS
LIN {X -87.4779,Y 69.5338,Z 115,A 138.5902,B 24.9319,C -1.9062,E1 24.872,E2 307.083} C_DIS
LIN {X -91.194,Y 64.5836,Z 115,A 140.5671,B 24.9358,C -1.8501,E1 24.8689,E2 305.2303} C_DIS
LIN {X -93.6118,Y 61.0245,Z 115,A 143.1768,B 24.9352,C -1.8597,E1 24.8648,E2 302.5846} C_DIS
LIN {X -97.0136,Y 55.4586,Z 115,A 146.1991,B 24.9367,C -1.8374,E1 24.8606,E2 299.5999} C_DIS
LIN {X -98.27,Y 53.2001,Z 115,A 147.6301,B 24.9367,C -1.8376,E1 24.8586,E2 298.1607} C_DIS
LIN {X -99.8607,Y 50.1539,Z 115,A 149.386,B 24.9371,C -1.8321,E1 24.8564,E2 296.4086} C_DIS
LIN {X -101.2223,Y 47.3427,Z 115,A 150.9936,B 24.9374,C -1.8275,E1 24.8545,E2 294.8032} C_DIS
LIN {X -103.8665,Y 41.2207,Z 115,A 154.4873,B 24.9379,C -1.8199,E1 24.8507,E2 291.3083} C_DIS
LIN {X -105.0121,Y 38.2061,Z 115,A 156.0764,B 24.9384,C -1.8122,E1 24.8491,E2 289.7286} C_DIS
LIN {X -106.104,Y 35.0654,Z 115,A 158.5926,B 24.9366,C -1.8386,E1 24.8469,E2 287.1351} C_DIS
LIN {X -107.491,Y 30.5437,Z 115,A 160.2653,B 24.9392,C -1.8015,E1 24.8456,E2 285.5412} C_DIS
LIN {X -108.9136,Y 25.0017,Z 115,A 163.2879,B 24.9396,C -1.7955,E1 24.8436,E2 282.5152} C_DIS
LIN {X -110.4239,Y 17.1406,Z 115,A 167.4142,B 24.9404,C -1.783,E1 24.8415,E2 278.3942} C_DIS
LIN {X -110.9188,Y 13.5868,Z 115,A 169.3964,B 24.9404,C -1.7826,E1 24.8408,E2 276.4013} C_DIS
LIN {X -111.3267,Y 9.6918,Z 115,A 171.1882,B 24.9414,C -1.7677,E1 24.8403,E2 274.6343} C_DIS
LIN {X -111.5619,Y 6.4221,Z 115,A 172.9561,B 24.9416,C -1.7656,E1 24.84,E2 272.8606} C_DIS
LIN {X -111.6982,Y 3.28,Z 115,A 174.5693,B 24.9419,C -1.7604,E1 24.8398,E2 271.2501} C_DIS
LIN {X -111.7445,Y -0.6266,Z 115,A 176.5533,B 24.9424,C -1.7532,E1 24.8398,E2 269.2715} C_DIS
LIN {X -111.695,Y -3.3864,Z 115,A 177.9767,B 24.9427,C -1.7489,E1 24.8398,E2 267.8497} C_DIS
LIN {X -111.5463,Y -6.7048,Z 115,A 179.8344,B 24.9427,C -1.7494,E1 24.8402,E2 265.9796} C_DIS
LIN {X -111.2767,Y -10.2336,Z 115,A -178.4971,B 24.9434,C -1.7379,E1 24.8406,E2 264.3286} C_DIS
LIN {X -110.9674,Y -13.1716,Z 115,A -176.9299,B 24.9436,C -1.7351,E1 24.8411,E2 262.7587} C_DIS
LIN {X -110.4623,Y -16.892,Z 115,A -174.7657,B 24.9434,C -1.7383,E1 24.8419,E2 260.5738} C_DIS
LIN {X -109.5742,Y -21.9327,Z 115,A -172.2594,B 24.9442,C -1.7254,E1 24.8432,E2 258.0836} C_DIS
LIN {X -108.2119,Y -27.8825,Z 115,A -169.2154,B 24.9451,C -1.7123,E1 24.8452,E2 255.0529} C_DIS
LIN {X -106.7758,Y -32.9573,Z 115,A -166.7832,B 24.9463,C -1.6934,E1 24.847,E2 252.6517} C_DIS
LIN {X -105.163,Y -37.7922,Z 115,A -163.9704,B 24.9463,C -1.6933,E1 24.8496,E2 249.8231} C_DIS
LIN {X -103.7724,Y -41.4602,Z 115,A -161.6999,B 24.946,C -1.6975,E1 24.8519,E2 247.5298} C_DIS
LIN {X -102.3974,Y -44.744,Z 115,A -159.8779,B 24.9463,C -1.6921,E1 24.8539,E2 245.7105} C_DIS
LIN {X -100.657,Y -48.5327,Z 115,A -157.8278,B 24.9469,C -1.6826,E1 24.8563,E2 243.672} C_DIS
LIN {X -98.7203,Y -52.3608,Z 115,A -155.5634,B 24.9472,C -1.679,E1 24.8592,E2 241.404} C_DIS
LIN {X -96.8549,Y -55.7347,Z 115,A -153.6615,B 24.9477,C -1.6707,E1 24.8618,E2 239.512} C_DIS
LIN {X -95.4532,Y -58.1028,Z 115,A -152.1707,B 24.9477,C -1.6701,E1 24.8639,E2 238.015} C_DIS
LIN {X -92.7596,Y -62.3142,Z 115,A -149.8171,B 24.9487,C -1.6551,E1 24.8675,E2 235.6852} C_DIS
LIN {X -90.5259,Y -65.5185,Z 115,A -146.953,B 24.9468,C -1.6845,E1 24.8723,E2 232.737} C_DIS
LIN {X -87.8829,Y -69.0213,Z 115,A -145.5724,B 24.9493,C -1.6442,E1 24.8745,E2 231.446} C_DIS
LIN {X -85.3589,Y -72.12,Z 115,A -142.6287,B 24.9474,C -1.6753,E1 24.8799,E2 228.4146} C_DIS
LIN {X -82.4412,Y -75.4368,Z 115,A -141.3237,B 24.9501,C -1.6315,E1 24.8822,E2 227.2081} C_DIS
LIN {X -80.5417,Y -77.4615,Z 115,A -139.5844,B 24.9495,C -1.641,E1 24.8856,E2 225.4386} C_DIS
LIN {X -78.0574,Y -79.967,Z 115,A -137.7522,B 24.9497,C -1.6381,E1 24.8892,E2 223.6057} C_DIS
LIN {X -75.5819,Y -82.3081,Z 115,A -135.9686,B 24.9498,C -1.636,E1 24.8928,E2 221.8197} C_DIS
LIN {X -72.3517,Y -85.1616,Z 115,A -133.7601,B 24.9501,C -1.6316,E1 24.8975,E2 219.613} C_DIS
LIN {X -69.2564,Y -87.6972,Z 115,A -131.8162,B 24.9506,C -1.6234,E1 24.9017,E2 217.6813} C_DIS
LIN {X -66.7385,Y -89.6294,Z 115,A -130.005,B 24.9503,C -1.628,E1 24.9058,E2 215.8526} C_DIS
LIN {X -61.4983,Y -93.3016,Z 115,A -126.768,B 24.9508,C -1.6208,E1 24.9132,E2 212.622} C_DIS
LIN {X -57.5834,Y -95.7688,Z 115,A -124.108,B 24.9503,C -1.629,E1 24.9196,E2 209.9341} C_DIS
LIN {X -53.3265,Y -98.2014,Z 115,A -121.9251,B 24.9513,C -1.6119,E1 24.9248,E2 207.7856} C_DIS
LIN {X -50.4875,Y -99.6916,Z 115,A -120.3232,B 24.9516,C -1.608,E1 24.9288,E2 206.1885} C_DIS
LIN {X -47.5312,Y -101.1345,Z 115,A -118.5602,B 24.9515,C -1.6091,E1 24.9332,E2 204.4183} C_DIS
LIN {X -44.6696,Y -102.4298,Z 115,A -116.9416,B 24.9515,C -1.6077,E1 24.9374,E2 202.7993} C_DIS
LIN {X -39.3362,Y -104.5943,Z 115,A -114.1066,B 24.952,C -1.5999,E1 24.9447,E2 199.9765} C_DIS
LIN {X -36.4532,Y -105.6349,Z 115,A -111.7091,B 24.95,C -1.6333,E1 24.9513,E2 197.4952} C_DIS
LIN {X -32.0611,Y -107.0486,Z 115,A -110.2919,B 24.9525,C -1.5916,E1 24.9548,E2 196.1745} C_DIS
LIN {X -30.0024,Y -107.6444,Z 115,A -108.8304,B 24.9517,C -1.6061,E1 24.9588,E2 194.6763} C_DIS
LIN {X -25.924,Y -108.6992,Z 115,A -106.8471,B 24.9522,C -1.5974,E1 24.9641,E2 192.7108} C_DIS
LIN {X -22.6834,Y -109.42,Z 115,A -105.0193,B 24.9519,C -1.6019,E1 24.9692,E2 190.87} C_DIS
LIN {X -19.4113,Y -110.0481,Z 115,A -103.4265,B 24.9522,C -1.5964,E1 24.9735,E2 189.2885} C_DIS
LIN {X -16.4509,Y -110.5305,Z 115,A -100.9035,B 24.9497,C -1.6382,E1 24.9808,E2 186.6644} C_DIS
LIN {X -10.8781,Y -111.2172,Z 115,A -99.0472,B 24.9524,C -1.5939,E1 24.9856,E2 184.912} C_DIS
LIN {X -6.939,Y -111.5323,Z 115,A -96.443,B 24.9509,C -1.6187,E1 24.993,E2 182.2481} C_DIS
LIN {X -3.3361,Y -111.6965,Z 115,A -95.3165,B 24.9528,C -1.5879,E1 24.996,E2 181.1944} C_DIS
LIN {X 0.7815,Y -111.721,Z 115,A -93.7405,B 24.9541,C -1.5658,E1 25.0003,E2 179.6707} C_DIS
Enddeposition()
LIN {X 0.7815,Y -111.721,Z 115,A -93.7405,B 24.9541,C -1.5658,E1 25.0003,E2 179.6707} C_DIS
Startdeposition()
$VEL.CP = VEL_PRINT
LIN {X -1.6781,Y -110.8211,Z 115,A -94.9942,B 24.9531,C -1.582,E1 24.9968,E2 180.886} C_DIS
LIN {X -5.5488,Y -110.6957,Z 115,A -97.1121,B 24.9534,C -1.5769,E1 24.9909,E2 183.0163} C_DIS
LIN {X -8.9868,Y -110.4684,Z 115,A -98.7943,B 24.9532,C -1.5811,E1 24.9862,E2 184.6894} C_DIS
LIN {X -11.2552,Y -110.2607,Z 115,A -100.5144,B 24.9545,C -1.5588,E1 24.9813,E2 186.4635} C_DIS
LIN {X -15.1164,Y -109.7986,Z 115,A -102.0751,B 24.9534,C -1.5777,E1 24.9771,E2 187.9804} C_DIS
LIN {X -18.7009,Y -109.245,Z 115,A -103.9623,B 24.9534,C -1.5777,E1 24.9719,E2 189.8692} C_DIS
LIN {X -22.4006,Y -108.546,Z 115,A -105.8227,B 24.9531,C -1.5821,E1 24.9668,E2 191.7215} C_DIS
LIN {X -26.0795,Y -107.7214,Z 115,A -107.8587,B 24.9533,C -1.5795,E1 24.9613,E2 193.7663} C_DIS
LIN {X -30.0134,Y -106.6923,Z 115,A -109.8912,B 24.953,C -1.5837,E1 24.9558,E2 195.792} C_DIS
LIN {X -36.3269,Y -104.7116,Z 115,A -113.111,B 24.9524,C -1.5945,E1 24.9473,E2 198.9918} C_DIS
LIN {X -41.4159,Y -102.8051,Z 115,A -116.1637,B 24.9528,C -1.5872,E1 24.9393,E2 202.0683} C_DIS
LIN {X -44.4968,Y -101.5091,Z 115,A -117.9459,B 24.9528,C -1.5868,E1 24.9347,E2 203.8555} C_DIS
LIN {X -48.0298,Y -99.8857,Z 115,A -119.8876,B 24.9525,C -1.5919,E1 24.9298,E2 205.7899} C_DIS
LIN {X -51.2168,Y -98.2908,Z 115,A -121.7787,B 24.9525,C -1.5923,E1 24.9251,E2 207.6853} C_DIS
LIN {X -54.3295,Y -96.6045,Z 115,A -123.7688,B 24.9527,C -1.5884,E1 24.9202,E2 209.6903} C_DIS
LIN {X -57.2837,Y -94.8825,Z 115,A -125.4564,B 24.9524,C -1.5942,E1 24.9162,E2 211.3693} C_DIS
LIN {X -60.8337,Y -92.6462,Z 115,A -127.8532,B 24.9527,C -1.5886,E1 24.9105,E2 213.7873} C_DIS
LIN {X -66.0551,Y -89.0008,Z 115,A -130.9087,B 24.9518,C -1.6035,E1 24.9036,E2 216.8178} C_DIS
LIN {X -68.4218,Y -87.193,Z 115,A -132.4984,B 24.9518,C -1.6043,E1 24.9001,E2 218.4115} C_DIS
LIN {X -71.6022,Y -84.6006,Z 115,A -134.6211,B 24.9515,C -1.6083,E1 24.8955,E2 220.5327} C_DIS
LIN {X -74.7499,Y -81.8323,Z 115,A -136.6396,B 24.9509,C -1.6185,E1 24.8914,E2 222.5351} C_DIS
LIN {X -76.767,Y -79.943,Z 115,A -138.1164,B 24.9509,C -1.6196,E1 24.8884,E2 224.0155} C_DIS
LIN {X -79.2359,Y -77.4983,Z 115,A -140.0211,B 24.9509,C -1.6191,E1 24.8846,E2 225.9293} C_DIS
Enddeposition()
END
